C05454=1097.638,130.250,436.850,176.760,16.481,152.162
C05455=1097.644,130.499,436.829,176.762,16.481,152.162
C05456=1097.649,130.749,436.810,176.765,16.482,152.161
C05457=1097.656,130.998,436.790,176.768,16.482,152.161
C05458=1097.661,131.248,436.771,176.771,16.482,152.160
C05459=1097.667,131.496,436.751,176.774,16.482,152.159
C05460=1097.673,131.745,436.730,176.777,16.482,152.159
C05461=1097.678,131.995,436.711,176.780,16.482,152.158
C05462=1097.684,132.244,436.691,176.783,16.483,152.158
C05463=1097.690,132.493,436.671,176.785,16.483,152.157
C05464=1097.695,132.742,436.651,176.789,16.483,152.157
C05465=1097.701,132.991,436.631,176.792,16.484,152.156
C05466=1097.706,133.241,436.611,176.794,16.484,152.156
C05467=1097.712,133.490,436.591,176.798,16.484,152.155
C05468=1097.718,133.738,436.571,176.801,16.484,152.155
C05469=1097.724,133.988,436.551,176.803,16.485,152.154
C05470=1097.729,134.237,436.532,176.806,16.485,152.154
C05471=1097.734,134.486,436.511,176.810,16.485,152.153
C05472=1097.740,134.735,436.491,176.812,16.485,152.152
C05473=1097.746,134.984,436.472,176.815,16.485,152.152
C05474=1097.751,135.234,436.451,176.819,16.486,152.151
C05475=1097.757,135.482,436.431,176.821,16.486,152.151
C05476=1097.763,135.731,436.411,176.824,16.486,152.150
C05477=1097.768,135.981,436.392,176.828,16.486,152.150
C05478=1097.774,136.230,436.371,176.830,16.486,152.149
C05479=1097.780,136.479,436.351,176.833,16.487,152.149
C05480=1097.786,136.728,436.331,176.836,16.487,152.148
C05481=1097.791,136.977,436.311,176.839,16.487,152.147
C05482=1097.797,137.226,436.291,176.842,16.488,152.147
C05483=1097.802,137.475,436.271,176.845,16.488,152.146
C05484=1097.808,137.724,436.251,176.848,16.488,152.146
C05485=1097.814,137.974,436.230,176.851,16.488,152.145
C05486=1097.820,138.223,436.210,176.854,16.489,152.145
C05487=1097.825,138.472,436.189,176.857,16.488,152.144
C05488=1097.831,138.721,436.169,176.860,16.489,152.143
C05489=1097.836,138.970,436.150,176.863,16.489,152.143
C05490=1097.842,139.219,436.130,176.866,16.489,152.142
C05491=1097.847,139.468,436.109,176.869,16.489,152.142
C05492=1097.853,139.717,436.089,176.872,16.490,152.141
C05493=1097.858,139.966,436.069,176.875,16.489,152.141
C05494=1097.864,140.216,436.048,176.878,16.490,152.140
C05495=1097.870,140.465,436.028,176.881,16.490,152.139
C05496=1097.875,140.714,436.007,176.884,16.490,152.139
C05497=1097.881,140.963,435.987,176.887,16.490,152.138
C05498=1097.887,141.212,435.967,176.890,16.490,152.138
C05499=1097.892,141.461,435.946,176.893,16.490,152.137
C05500=1097.898,141.710,435.926,176.896,16.491,152.137
C05501=1097.903,141.959,435.906,176.899,16.491,152.136
C05502=1097.909,142.209,435.885,176.902,16.491,152.135
C05503=1097.915,142.458,435.865,176.905,16.491,152.135
C05504=1097.920,142.707,435.844,176.908,16.492,152.134
C05505=1097.926,142.956,435.824,176.912,16.492,152.134
C05506=1097.932,143.205,435.804,176.914,16.492,152.133
C05507=1097.937,143.454,435.783,176.917,16.492,152.133
C05508=1097.944,143.729,435.760,176.921,16.492,152.132
C05509=1097.950,144.003,435.738,176.924,16.492,152.131
C05510=1097.956,144.278,435.714,176.928,16.492,152.130
C05511=1097.962,144.552,435.692,176.931,16.493,152.130
C05512=1097.967,144.801,435.671,176.934,16.493,152.129
C05513=1097.973,145.050,435.652,176.937,16.493,152.129
C05514=1097.979,145.300,435.631,176.940,16.493,152.128
C05515=1097.985,145.549,435.610,176.943,16.493,152.128
C05516=1097.990,145.798,435.590,176.946,16.493,152.127
C05517=1097.996,146.046,435.569,176.949,16.493,152.126
C05518=1098.001,146.295,435.548,176.953,16.494,152.126
C05519=1098.007,146.545,435.527,176.955,16.493,152.125
C05520=1098.013,146.794,435.507,176.959,16.494,152.125
C05521=1098.019,147.043,435.487,176.962,16.494,152.124
C05522=1098.024,147.291,435.466,176.964,16.494,152.123
C05523=1098.030,147.541,435.445,176.968,16.494,152.123
C05524=1098.035,147.790,435.424,176.971,16.494,152.122
C05525=1098.041,148.039,435.404,176.974,16.494,152.122
C05526=1098.047,148.288,435.383,176.977,16.494,152.121
C05527=1098.053,148.537,435.362,176.980,16.494,152.120
C05528=1098.058,148.787,435.341,176.984,16.495,152.120
C05529=1098.063,149.035,435.320,176.986,16.494,152.119
C05530=1098.069,149.285,435.299,176.989,16.495,152.119
C05531=1098.075,149.534,435.279,176.993,16.495,152.118
C05532=1098.081,149.782,435.258,176.995,16.495,152.117
C05533=1098.086,150.031,435.237,176.999,16.495,152.117
C05534=1098.092,150.281,435.217,177.002,16.495,152.116
C05535=1098.097,150.530,435.195,177.005,16.495,152.115
C05536=1098.103,150.779,435.175,177.008,16.495,152.115
C05537=1098.108,151.028,435.154,177.012,16.495,152.114
C05538=1098.114,151.277,435.132,177.015,16.496,152.114
C05539=1098.119,151.526,435.112,177.017,16.495,152.113
C05540=1098.125,151.775,435.091,177.021,16.496,152.112
C05541=1098.131,152.025,435.070,177.024,16.496,152.112
C05542=1098.137,152.273,435.049,177.027,16.495,152.111
C05543=1098.142,152.522,435.029,177.030,16.495,152.110
C05544=1098.148,152.772,435.008,177.033,16.496,152.110
C05545=1098.154,153.020,434.986,177.037,16.496,152.109
C05546=1098.159,153.269,434.966,177.039,16.496,152.109
C05547=1098.165,153.519,434.944,177.043,16.496,152.108
C05548=1098.170,153.768,434.924,177.046,16.496,152.107
C05549=1098.176,154.016,434.902,177.049,16.496,152.107
C05550=1098.182,154.266,434.881,177.052,16.496,152.106
C05551=1098.187,154.515,434.860,177.055,16.496,152.105
C05552=1098.193,154.763,434.839,177.059,16.496,152.105
C05553=1098.199,155.013,434.818,177.061,16.496,152.104
C05554=1098.204,155.261,434.797,177.065,16.496,152.104
C05555=1098.210,155.511,434.776,177.068,16.497,152.103
C05556=1098.216,155.760,434.754,177.071,16.496,152.102
C05557=1098.221,156.009,434.734,177.074,16.496,152.102
C05558=1098.227,156.258,434.712,177.078,16.496,152.101
C05559=1098.232,156.507,434.690,177.081,16.497,152.100
C05560=1098.238,156.757,434.670,177.084,16.496,152.100
C05561=1098.244,157.005,434.648,177.087,16.497,152.099
C05562=1098.249,157.254,434.627,177.090,16.496,152.098
C05563=1098.255,157.504,434.606,177.094,16.497,152.098
C05564=1098.261,157.752,434.585,177.096,16.496,152.097
C05565=1098.267,158.001,434.563,177.100,16.497,152.097
C05566=1098.272,158.250,434.543,177.103,16.497,152.096
C05567=1098.277,158.499,434.521,177.106,16.496,152.095
C05568=1098.283,158.748,434.499,177.109,16.496,152.095
C05569=1098.288,158.997,434.479,177.112,16.497,152.094
C05570=1098.294,159.247,434.457,177.116,16.497,152.093
C05571=1098.300,159.495,434.436,177.118,16.497,152.093
C05572=1098.306,159.770,434.412,177.122,16.497,152.092
C05573=1098.312,160.044,434.389,177.126,16.496,152.091
C05574=1098.319,160.318,434.365,177.129,16.496,152.091
C05575=1098.325,160.592,434.341,177.133,16.496,152.090
C05576=1098.331,160.842,434.320,177.136,16.496,152.089
C05577=1098.335,161.090,434.299,177.139,16.497,152.089
C05578=1098.342,161.340,434.277,177.143,16.497,152.088
C05579=1098.347,161.588,434.256,177.146,16.497,152.087
C05580=1098.353,161.837,434.234,177.149,16.496,152.087
C05581=1098.358,162.086,434.212,177.152,16.497,152.086
C05582=1098.364,162.336,434.191,177.156,16.497,152.085
C05583=1098.370,162.585,434.170,177.158,16.497,152.085
C05584=1098.374,162.833,434.148,177.162,16.497,152.084
C05585=1098.381,163.083,434.126,177.165,16.497,152.083
C05586=1098.385,163.331,434.105,177.169,16.497,152.083
C05587=1098.392,163.581,434.083,177.171,16.496,152.082
C05588=1098.396,163.829,434.061,177.175,16.497,152.081
C05589=1098.403,164.079,434.039,177.178,16.497,152.081
C05590=1098.408,164.327,434.018,177.181,16.497,152.080
C05591=1098.413,164.577,433.996,177.184,16.497,152.079
C05592=1098.419,164.825,433.975,177.188,16.497,152.079
C05593=1098.424,165.074,433.953,177.191,16.497,152.078
C05594=1098.430,165.323,433.931,177.195,16.497,152.077
C05595=1098.435,165.572,433.909,177.198,16.497,152.077
C05596=1098.441,165.821,433.888,177.201,16.497,152.076
C05597=1098.446,166.070,433.866,177.204,16.497,152.075
C05598=1098.452,166.319,433.844,177.207,16.497,152.075
C05599=1098.457,166.568,433.822,177.211,16.497,152.074
C05600=1098.463,166.817,433.801,177.214,16.496,152.073
C05601=1098.469,167.066,433.779,177.217,16.497,152.073
C05602=1098.474,167.315,433.757,177.221,16.497,152.072
C05603=1098.480,167.564,433.736,177.224,16.497,152.071
C05604=1098.485,167.813,433.714,177.227,16.497,152.071
C05605=1098.491,168.062,433.692,177.230,16.497,152.070
C05606=1098.496,168.311,433.670,177.234,16.497,152.069
C05607=1098.502,168.560,433.649,177.237,16.497,152.069
C05608=1098.507,168.809,433.626,177.240,16.496,152.068
C05609=1098.513,169.058,433.604,177.243,16.496,152.067
C05610=1098.519,169.307,433.582,177.247,16.496,152.067
C05611=1098.524,169.556,433.560,177.250,16.497,152.066
C05612=1098.530,169.805,433.539,177.254,16.497,152.065
C05613=1098.535,170.054,433.517,177.256,16.496,152.065
C05614=1098.541,170.303,433.494,177.260,16.496,152.064
C05615=1098.546,170.552,433.473,177.263,16.496,152.063
C05616=1098.552,170.801,433.451,177.267,16.496,152.063
C05617=1098.558,171.050,433.429,177.269,16.496,152.062
C05618=1098.563,171.298,433.407,177.273,16.496,152.061
C05619=1098.569,171.548,433.384,177.276,16.496,152.061
C05620=1098.574,171.797,433.362,177.280,16.496,152.060
C05621=1098.580,172.046,433.341,177.283,16.496,152.059
C05622=1098.586,172.295,433.318,177.286,16.495,152.059
C05623=1098.592,172.544,433.296,177.290,16.495,152.058
C05624=1098.597,172.793,433.274,177.293,16.495,152.057
C05625=1098.602,173.042,433.252,177.297,16.495,152.056
C05626=1098.608,173.291,433.230,177.299,16.495,152.056
C05627=1098.613,173.540,433.208,177.303,16.495,152.055
C05628=1098.620,173.788,433.186,177.306,16.495,152.054
C05629=1098.625,174.038,433.163,177.310,16.495,152.054
C05630=1098.630,174.287,433.142,177.313,16.495,152.053
C05631=1098.636,174.535,433.119,177.316,16.495,152.052
C05632=1098.642,174.785,433.097,177.320,16.495,152.052
C05633=1098.647,175.033,433.074,177.323,16.494,152.051
C05634=1098.653,175.282,433.053,177.327,16.494,152.050
C05635=1098.659,175.532,433.031,177.329,16.494,152.049
C05636=1098.665,175.805,433.006,177.334,16.494,152.049
C05637=1098.671,176.079,432.981,177.338,16.494,152.048
C05638=1098.678,176.353,432.957,177.341,16.494,152.047
C05639=1098.683,176.626,432.932,177.345,16.493,152.046
C05640=1098.689,176.876,432.911,177.349,16.493,152.045
C05641=1098.695,177.124,432.888,177.351,16.493,152.045
C05642=1098.700,177.374,432.865,177.355,16.493,152.044
C05643=1098.707,177.623,432.843,177.358,16.493,152.043
C05644=1098.712,177.871,432.820,177.362,16.493,152.043
C05645=1098.718,178.120,432.798,177.365,16.492,152.042
C05646=1098.723,178.369,432.775,177.368,16.492,152.041
C05647=1098.729,178.618,432.754,177.372,16.492,152.040
C05648=1098.735,178.867,432.731,177.375,16.492,152.040
C05649=1098.740,179.116,432.709,177.379,16.492,152.039
C05650=1098.746,179.365,432.686,177.382,16.491,152.038
C05651=1098.752,179.614,432.664,177.385,16.491,152.038
C05652=1098.758,179.863,432.641,177.389,16.491,152.037
C05653=1098.763,180.112,432.618,177.392,16.491,152.036
C05654=1098.770,180.361,432.596,177.396,16.491,152.035
C05655=1098.775,180.609,432.574,177.399,16.490,152.035
C05656=1098.780,180.858,432.551,177.402,16.490,152.034
C05657=1098.786,181.107,432.528,177.406,16.490,152.033
C05658=1098.792,181.356,432.507,177.410,16.490,152.032
C05659=1098.798,181.605,432.484,177.413,16.490,152.032
C05660=1098.804,181.854,432.461,177.416,16.490,152.031
C05661=1098.809,182.103,432.438,177.420,16.489,152.030
C05662=1098.814,182.352,432.416,177.423,16.489,152.029
C05663=1098.821,182.600,432.394,177.427,16.489,152.029
C05664=1098.826,182.849,432.371,177.430,16.489,152.028
C05665=1098.832,183.098,432.348,177.433,16.489,152.027
C05666=1098.838,183.348,432.325,177.437,16.488,152.026
C05667=1098.843,183.597,432.302,177.440,16.488,152.026
C05668=1098.850,183.845,432.280,177.444,16.488,152.025
C05669=1098.856,184.094,432.257,177.448,16.488,152.024
C05670=1098.861,184.343,432.234,177.451,16.487,152.023
C05671=1098.867,184.592,432.211,177.454,16.487,152.023
C05672=1098.872,184.841,432.189,177.458,16.487,152.022
C05673=1098.878,185.090,432.166,177.461,16.487,152.021
C05674=1098.884,185.339,432.143,177.465,16.487,152.020
C05675=1098.889,185.587,432.121,177.469,16.487,152.020
C05676=1098.895,185.836,432.098,177.471,16.486,152.019
C05677=1098.900,186.085,432.075,177.475,16.486,152.018
C05678=1098.906,186.334,432.052,177.478,16.486,152.017
C05679=1098.912,186.583,432.029,177.482,16.486,152.017
C05680=1098.918,186.832,432.006,177.486,16.486,152.016
C05681=1098.923,187.081,431.983,177.489,16.486,152.015
C05682=1098.927,187.330,431.960,177.492,16.485,152.015
C05683=1098.933,187.579,431.938,177.496,16.485,152.014
C05684=1098.939,187.828,431.915,177.499,16.485,152.013
C05685=1098.945,188.077,431.892,177.503,16.485,152.012
C05686=1098.950,188.326,431.869,177.506,16.485,152.012
C05687=1098.956,188.574,431.846,177.510,16.485,152.011
C05688=1098.961,188.824,431.822,177.513,16.484,152.010
C05689=1098.967,189.073,431.799,177.516,16.484,152.009
C05690=1098.973,189.321,431.776,177.520,16.484,152.009
C05691=1098.979,189.570,431.753,177.523,16.484,152.008
C05692=1098.984,189.818,431.730,177.527,16.484,152.007
C05693=1098.989,190.067,431.707,177.531,16.483,152.006
C05694=1098.994,190.316,431.684,177.534,16.483,152.006
C05695=1099.000,190.565,431.661,177.537,16.483,152.005
C05696=1099.006,190.814,431.638,177.541,16.483,152.004
C05697=1099.012,191.063,431.615,177.545,16.482,152.003
C05698=1099.017,191.312,431.591,177.548,16.482,152.003
C05699=1099.022,191.561,431.568,177.552,16.482,152.002
C05700=1099.029,191.834,431.542,177.555,16.482,152.001
C05701=1099.035,192.108,431.517,177.559,16.482,152.000
C05702=1099.041,192.381,431.491,177.563,16.482,151.999
C05703=1099.047,192.654,431.465,177.567,16.481,151.998
C05704=1099.053,192.903,431.443,177.570,16.481,151.998
C05705=1099.059,193.152,431.420,177.574,16.481,151.997
C05706=1099.064,193.401,431.396,177.578,16.481,151.996
C05707=1099.070,193.650,431.373,177.581,16.481,151.995
C05708=1099.076,193.899,431.349,177.584,16.480,151.995
C05709=1099.081,194.147,431.326,177.588,16.480,151.994
C05710=1099.086,194.397,431.303,177.591,16.480,151.993
C05711=1099.092,194.645,431.279,177.595,16.479,151.992
C05712=1099.098,194.894,431.256,177.599,16.479,151.992
C05713=1099.103,195.143,431.233,177.602,16.479,151.991
C05714=1099.109,195.391,431.209,177.606,16.479,151.990
C05715=1099.115,195.641,431.186,177.609,16.478,151.989
C05716=1099.120,195.890,431.162,177.613,16.478,151.988
C05717=1099.126,196.138,431.139,177.616,16.478,151.988
C05718=1099.132,196.387,431.116,177.620,16.478,151.987
C05719=1099.137,196.637,431.092,177.623,16.477,151.986
C05720=1099.143,196.885,431.068,177.627,16.478,151.985
C05721=1099.149,197.134,431.046,177.631,16.477,151.984
C05722=1099.154,197.382,431.021,177.634,16.477,151.984
C05723=1099.160,197.631,430.998,177.637,16.476,151.983
C05724=1099.166,197.881,430.975,177.641,16.476,151.982
C05725=1099.172,198.129,430.951,177.645,16.476,151.981
C05726=1099.177,198.378,430.928,177.648,16.476,151.981
C05727=1099.183,198.627,430.904,177.652,16.475,151.980
C05728=1099.188,198.876,430.881,177.656,16.475,151.979
C05729=1099.194,199.124,430.857,177.660,16.475,151.978
C05730=1099.199,199.373,430.833,177.662,16.474,151.977
C05731=1099.206,199.622,430.809,177.666,16.474,151.977
C05732=1099.212,199.871,430.786,177.670,16.474,151.976
C05733=1099.217,200.120,430.762,177.674,16.473,151.975
C05734=1099.223,200.368,430.739,177.677,16.473,151.974
C05735=1099.228,200.617,430.715,177.681,16.473,151.973
C05736=1099.235,200.866,430.691,177.684,16.473,151.973
C05737=1099.240,201.115,430.668,177.688,16.473,151.972
C05738=1099.246,201.364,430.644,177.691,16.472,151.971
C05739=1099.252,201.612,430.620,177.695,16.472,151.970
C05740=1099.257,201.862,430.596,177.699,16.471,151.969
C05741=1099.263,202.110,430.573,177.702,16.471,151.969
C05742=1099.269,202.359,430.548,177.706,16.471,151.968
C05743=1099.274,202.608,430.525,177.710,16.470,151.967
C05744=1099.280,202.856,430.501,177.713,16.470,151.966
C05745=1099.286,203.105,430.477,177.717,16.470,151.965
C05746=1099.291,203.354,430.453,177.720,16.469,151.965
C05747=1099.297,203.603,430.430,177.724,16.469,151.964
C05748=1099.303,203.851,430.406,177.727,16.469,151.963
C05749=1099.308,204.100,430.382,177.731,16.469,151.962
C05750=1099.314,204.349,430.358,177.735,16.469,151.962
C05751=1099.320,204.598,430.334,177.739,16.468,151.961
C05752=1099.325,204.847,430.309,177.742,16.468,151.960
C05753=1099.331,205.095,430.287,177.746,16.468,151.959
C05754=1099.337,205.345,430.262,177.750,16.468,151.958
C05755=1099.342,205.593,430.238,177.753,16.467,151.957
C05756=1099.348,205.842,430.214,177.756,16.466,151.957
C05757=1099.353,206.090,430.190,177.760,16.466,151.956
C05758=1099.359,206.340,430.166,177.764,16.466,151.955
C05759=1099.365,206.588,430.142,177.767,16.466,151.954
C05760=1099.370,206.837,430.118,177.771,16.466,151.953
C05761=1099.375,207.086,430.094,177.775,16.465,151.953
C05762=1099.382,207.335,430.070,177.778,16.465,151.952
C05763=1099.387,207.583,430.045,177.782,16.465,151.951
C05764=1099.410,208.592,429.948,177.824,16.478,151.946
C05765=1099.419,208.961,429.911,177.829,16.479,151.945
C05766=1099.427,209.331,429.875,177.833,16.480,151.944
C05767=1099.436,209.701,429.839,177.839,16.480,151.943
C05768=1099.444,210.070,429.803,177.844,16.482,151.942
C05769=1099.450,210.320,429.778,177.847,16.482,151.941
C05770=1099.455,210.568,429.754,177.851,16.482,151.941
C05771=1099.461,210.818,429.729,177.855,16.483,151.940
C05772=1099.466,211.066,429.704,177.858,16.484,151.940
C05773=1099.472,211.314,429.680,177.861,16.484,151.939
C05774=1099.478,211.563,429.656,177.864,16.485,151.939
C05775=1099.483,211.812,429.631,177.868,16.485,151.938
C05776=1099.489,212.061,429.607,177.872,16.486,151.938
C05777=1099.494,212.309,429.582,177.875,16.486,151.937
C05778=1099.500,212.558,429.557,177.878,16.487,151.936
C05779=1099.506,212.807,429.533,177.882,16.487,151.936
C05780=1099.511,213.056,429.509,177.885,16.488,151.935
C05781=1099.517,213.304,429.483,177.889,16.489,151.935
C05782=1099.522,213.553,429.459,177.892,16.489,151.934
C05783=1099.528,213.802,429.434,177.895,16.490,151.934
C05784=1099.534,214.051,429.410,177.899,16.490,151.933
C05785=1099.539,214.299,429.385,177.903,16.492,151.932
C05786=1099.545,214.548,429.361,177.906,16.492,151.932
C05787=1099.550,214.797,429.336,177.909,16.493,151.931
C05788=1099.557,215.045,429.311,177.912,16.493,151.931
C05789=1099.561,215.294,429.286,177.916,16.494,151.930
C05790=1099.567,215.543,429.261,177.920,16.494,151.930
C05791=1099.573,215.792,429.236,177.923,16.495,151.929
C05792=1099.579,216.041,429.212,177.926,16.495,151.928
C05793=1099.584,216.289,429.187,177.930,16.496,151.928
C05794=1099.590,216.538,429.162,177.934,16.497,151.927
C05795=1099.596,216.786,429.137,177.937,16.497,151.927
C05796=1099.601,217.036,429.112,177.940,16.498,151.926
C05797=1099.606,217.284,429.087,177.943,16.498,151.926
C05798=1099.612,217.533,429.062,177.947,16.499,151.925
C05799=1099.618,217.782,429.038,177.951,16.500,151.925
C05800=1099.624,218.030,429.013,177.954,16.500,151.924
C05801=1099.628,218.279,428.988,177.957,16.501,151.923
C05802=1099.635,218.528,428.963,177.961,16.502,151.923
C05803=1099.640,218.776,428.938,177.965,16.502,151.922
C05804=1099.646,219.025,428.913,177.968,16.503,151.922
C05805=1099.652,219.273,428.888,177.971,16.503,151.921
C05806=1099.657,219.523,428.863,177.975,16.504,151.921
C05807=1099.663,219.771,428.838,177.978,16.505,151.920
C05808=1099.668,220.020,428.813,177.982,16.505,151.919
C05809=1099.675,220.269,428.788,177.985,16.506,151.919
C05810=1099.679,220.517,428.762,177.989,16.507,151.918
C05811=1099.685,220.766,428.738,177.992,16.507,151.918
C05812=1099.692,221.015,428.712,177.995,16.508,151.917
C05813=1099.697,221.263,428.687,177.999,16.508,151.917
C05814=1099.702,221.512,428.662,178.003,16.509,151.916
C05815=1099.708,221.760,428.637,178.006,16.510,151.915
C05816=1099.714,222.009,428.612,178.009,16.510,151.915
C05817=1099.723,222.383,428.574,178.014,16.511,151.914
C05818=1099.731,222.757,428.536,178.020,16.512,151.913
C05819=1099.739,223.131,428.499,178.025,16.514,151.913
C05820=1099.748,223.504,428.460,178.030,16.514,151.912
C05821=1099.753,223.753,428.435,178.033,16.515,151.911
C05822=1099.759,224.001,428.410,178.037,16.516,151.910
C05823=1099.764,224.250,428.385,178.041,16.517,151.910
C05824=1099.770,224.498,428.359,178.044,16.517,151.909
C05825=1099.775,224.747,428.333,178.047,16.518,151.909
C05826=1099.781,224.995,428.308,178.051,16.519,151.908
C05827=1099.786,225.245,428.283,178.054,16.519,151.908
C05828=1099.792,225.494,428.258,178.058,16.520,151.907
C05829=1099.797,225.742,428.232,178.062,16.521,151.907
C05830=1099.804,225.991,428.207,178.065,16.521,151.906
C05831=1099.810,226.239,428.181,178.068,16.522,151.906
C05832=1099.815,226.487,428.156,178.071,16.522,151.905
C05833=1099.821,226.736,428.131,178.075,16.524,151.904
C05834=1099.826,226.985,428.105,178.079,16.524,151.904
C05835=1099.832,227.234,428.079,178.082,16.525,151.903
C05836=1099.837,227.482,428.054,178.086,16.526,151.903
C05837=1099.843,227.731,428.028,178.089,16.526,151.902
C05838=1099.849,227.980,428.002,178.093,16.526,151.902
C05839=1099.854,228.228,427.977,178.097,16.527,151.901
C05840=1099.860,228.477,427.952,178.100,16.528,151.900
C05841=1099.866,228.726,427.926,178.103,16.528,151.900
C05842=1099.872,228.974,427.900,178.107,16.530,151.899
C05843=1099.877,229.223,427.875,178.110,16.530,151.899
C05844=1099.883,229.471,427.849,178.114,16.531,151.898
C05845=1099.888,229.720,427.823,178.117,16.531,151.898
C05846=1099.895,229.969,427.798,178.121,16.532,151.897
C05847=1099.900,230.218,427.772,178.124,16.533,151.897
C05848=1099.905,230.466,427.747,178.127,16.533,151.896
C05849=1099.911,230.715,427.721,178.131,16.534,151.896
C05850=1099.917,230.963,427.695,178.135,16.535,151.895
C05851=1099.922,231.212,427.669,178.138,16.536,151.894
C05852=1099.928,231.460,427.644,178.142,16.537,151.894
C05853=1099.933,231.709,427.618,178.145,16.537,151.893
C05854=1099.939,231.958,427.592,178.148,16.538,151.893
C05855=1099.944,232.207,427.566,178.152,16.539,151.892
C05856=1099.951,232.455,427.540,178.156,16.539,151.892
C05857=1099.956,232.703,427.514,178.159,16.540,151.891
C05858=1099.961,232.952,427.488,178.163,16.541,151.891
C05859=1099.967,233.201,427.463,178.166,16.542,151.890
C05860=1099.973,233.449,427.436,178.169,16.542,151.890
C05861=1099.979,233.698,427.410,178.173,16.543,151.889
C05862=1099.984,233.947,427.385,178.176,16.544,151.888
C05863=1099.990,234.195,427.359,178.180,16.544,151.888
C05864=1099.995,234.444,427.333,178.184,16.545,151.887
C05865=1100.001,234.693,427.307,178.187,16.546,151.887
C05866=1100.007,234.941,427.280,178.191,16.547,151.886
C05867=1100.012,235.190,427.254,178.194,16.548,151.886
C05868=1100.018,235.439,427.228,178.197,16.549,151.885
C05869=1100.025,235.803,427.190,178.203,16.549,151.884
C05870=1100.034,236.169,427.152,178.208,16.551,151.884
C05871=1100.042,236.534,427.113,178.213,16.552,151.883
C05872=1100.050,236.899,427.075,178.218,16.553,151.882
C05873=1100.056,237.148,427.049,178.221,16.554,151.882
C05874=1100.062,237.396,427.023,178.225,16.555,151.881
C05875=1100.068,237.645,426.997,178.228,16.556,151.881
C05876=1100.074,237.893,426.970,178.232,16.557,151.880
C05877=1100.079,238.142,426.944,178.236,16.557,151.880
C05878=1100.084,238.390,426.918,178.239,16.558,151.879
C05879=1100.090,238.639,426.892,178.243,16.559,151.878
C05880=1100.096,238.887,426.866,178.246,16.559,151.878
C05881=1100.101,239.136,426.840,178.249,16.560,151.877
C05882=1100.107,239.384,426.813,178.253,16.561,151.877
C05883=1100.112,239.633,426.787,178.256,16.562,151.876
C05884=1100.118,239.882,426.760,178.260,16.563,151.876
C05885=1100.124,240.130,426.734,178.264,16.563,151.875
C05886=1100.129,240.379,426.708,178.267,16.564,151.875
C05887=1100.135,240.628,426.681,178.271,16.565,151.874
C05888=1100.141,240.877,426.655,178.274,16.566,151.874
C05889=1100.146,241.125,426.629,178.277,16.567,151.873
C05890=1100.152,241.373,426.602,178.281,16.568,151.873
C05891=1100.158,241.622,426.575,178.284,16.568,151.872
C05892=1100.163,241.871,426.549,178.288,16.569,151.872
C05893=1100.169,242.119,426.523,178.292,16.570,151.871
C05894=1100.175,242.367,426.496,178.295,16.570,151.870
C05895=1100.180,242.616,426.470,178.299,16.572,151.870
C05896=1100.186,242.865,426.443,178.302,16.572,151.869
C05897=1100.192,243.113,426.417,178.306,16.573,151.869
C05898=1100.198,243.361,426.390,178.309,16.574,151.868
C05899=1100.203,243.610,426.364,178.312,16.575,151.868
C05900=1100.209,243.859,426.338,178.316,16.576,151.867
C05901=1100.214,244.107,426.310,178.319,16.576,151.867
C05902=1100.220,244.356,426.284,178.323,16.578,151.866
C05903=1100.225,244.604,426.257,178.327,16.578,151.866
C05904=1100.231,244.852,426.230,178.331,16.579,151.865
C05905=1100.237,245.101,426.204,178.334,16.580,151.865
C05906=1100.242,245.350,426.177,178.337,16.581,151.864
C05907=1100.248,245.598,426.151,178.341,16.582,151.864
C05908=1100.253,245.847,426.124,178.344,16.583,151.863
C05909=1100.259,246.095,426.097,178.348,16.584,151.863
C05910=1100.265,246.344,426.070,178.351,16.585,151.862
C05911=1100.271,246.593,426.043,178.355,16.586,151.862
C05912=1100.276,246.841,426.016,178.358,16.586,151.861
C05913=1100.282,247.090,425.990,178.361,16.587,151.861
C05914=1100.288,247.338,425.963,178.365,16.588,151.860
C05915=1100.293,247.587,425.936,178.369,16.589,151.860
C05916=1100.299,247.835,425.909,178.372,16.590,151.859
C05917=1100.304,248.083,425.883,178.376,16.591,151.859
C05918=1100.309,248.332,425.855,178.380,16.592,151.858
C05919=1100.315,248.580,425.829,178.383,16.593,151.858
C05920=1100.320,248.829,425.801,178.387,16.594,151.857
C05921=1100.328,249.187,425.763,178.391,16.595,151.857
C05922=1100.337,249.545,425.724,178.396,16.596,151.856
C05923=1100.344,249.904,425.685,178.401,16.597,151.855
C05924=1100.353,250.263,425.646,178.406,16.599,151.854
C05925=1100.358,250.511,425.618,178.410,16.600,151.854
C05926=1100.364,250.760,425.592,178.413,16.601,151.853
C05927=1100.370,251.008,425.565,178.417,16.602,151.853
C05928=1100.375,251.256,425.537,178.420,16.603,151.852
C05929=1100.381,251.504,425.511,178.424,16.604,151.852
C05930=1100.386,251.753,425.483,178.427,16.605,151.851
C05931=1100.392,252.001,425.457,178.431,16.606,151.851
C05932=1100.397,252.251,425.429,178.434,16.607,151.850
C05933=1100.403,252.498,425.402,178.438,16.608,151.850
C05934=1100.408,252.747,425.374,178.441,16.609,151.849
C05935=1100.414,252.996,425.348,178.445,16.610,151.849
C05936=1100.419,253.244,425.321,178.449,16.610,151.848
C05937=1100.426,253.493,425.293,178.452,16.612,151.848
C05938=1100.431,253.741,425.266,178.456,16.613,151.847
C05939=1100.437,253.990,425.239,178.459,16.613,151.847
C05940=1100.442,254.238,425.211,178.462,16.615,151.847
C05941=1100.448,254.486,425.184,178.466,16.615,151.846
C05942=1100.454,254.735,425.156,178.470,16.616,151.845
C05943=1100.459,254.983,425.129,178.473,16.617,151.845
C05944=1100.464,255.232,425.102,178.477,16.619,151.845
C05945=1100.471,255.480,425.075,178.480,16.619,151.844
C05946=1100.476,255.729,425.047,178.484,16.620,151.843
C05947=1100.482,255.977,425.019,178.487,16.621,151.843
C05948=1100.487,256.225,424.992,178.491,16.622,151.843
C05949=1100.492,256.474,424.965,178.494,16.623,151.842
C05950=1100.499,256.722,424.938,178.498,16.624,151.841
C05951=1100.504,256.971,424.910,178.501,16.625,151.841
C05952=1100.510,257.219,424.883,178.505,16.626,151.841
C05953=1100.516,257.468,424.855,178.508,16.627,151.840
C05954=1100.521,257.716,424.827,178.512,16.629,151.840
C05955=1100.527,257.964,424.800,178.515,16.629,151.839
C05956=1100.532,258.213,424.773,178.519,16.630,151.839
C05957=1100.538,258.461,424.744,178.522,16.631,151.838
C05958=1100.544,258.710,424.718,178.526,16.632,151.838
C05959=1100.549,258.958,424.690,178.529,16.633,151.837
C05960=1100.556,259.206,424.662,178.533,16.634,151.837
C05961=1100.561,259.455,424.635,178.536,16.635,151.836
C05962=1100.566,259.703,424.607,178.540,16.636,151.836
C05963=1100.573,259.952,424.580,178.543,16.637,151.835
C05964=1100.578,260.200,424.552,178.547,16.638,151.835
C05965=1100.584,260.449,424.524,178.550,16.639,151.834
C05966=1100.590,260.697,424.496,178.554,16.640,151.834
C05967=1100.595,260.945,424.469,178.558,16.641,151.833
C05968=1100.601,261.194,424.441,178.561,16.642,151.833
C05969=1100.607,261.442,424.413,178.565,16.643,151.832
C05970=1100.613,261.691,424.386,178.569,16.644,151.832
C05971=1100.618,261.939,424.358,178.571,16.645,151.831
C05972=1100.623,262.187,424.330,178.575,16.646,151.831
C05973=1100.633,262.543,424.290,178.581,16.648,151.830
C05974=1100.640,262.898,424.251,178.586,16.649,151.829
C05975=1100.649,263.254,424.210,178.591,16.650,151.829
C05976=1100.657,263.609,424.171,178.596,16.652,151.828
C05977=1100.663,263.858,424.142,178.599,16.653,151.828
C05978=1100.669,264.105,424.115,178.603,16.654,151.827
C05979=1100.675,264.354,424.087,178.607,16.655,151.827
C05980=1100.680,264.602,424.059,178.610,16.656,151.826
C05981=1100.686,264.852,424.031,178.614,16.657,151.826
C05982=1100.691,265.100,424.003,178.617,16.658,151.825
C05983=1100.697,265.348,423.975,178.621,16.659,151.825
C05984=1100.702,265.596,423.947,178.623,16.660,151.824
C05985=1100.708,265.844,423.919,178.627,16.662,151.824
C05986=1100.713,266.093,423.891,178.631,16.663,151.823
C05987=1100.719,266.341,423.863,178.634,16.664,151.823
C05988=1100.725,266.590,423.834,178.638,16.665,151.823
C05989=1100.730,266.838,423.806,178.641,16.666,151.822
C05990=1100.736,267.087,423.778,178.645,16.668,151.822
C05991=1100.741,267.335,423.750,178.648,16.668,151.821
C05992=1100.747,267.584,423.722,178.652,16.670,151.821
C05993=1100.753,267.832,423.694,178.656,16.671,151.820
C05994=1100.759,268.080,423.665,178.659,16.672,151.820
C05995=1100.764,268.328,423.637,178.663,16.673,151.819
C05996=1100.770,268.577,423.608,178.666,16.674,151.819
C05997=1100.776,268.825,423.580,178.670,16.675,151.818
C05998=1100.781,269.073,423.552,178.673,16.676,151.818
C05999=1100.787,269.321,423.524,178.677,16.678,151.818
C06000=1100.793,269.570,423.496,178.680,16.679,151.817
C06001=1100.798,269.818,423.467,178.684,16.680,151.817
C06002=1100.804,270.066,423.439,178.687,16.681,151.816
C06003=1100.810,270.314,423.411,178.691,16.682,151.816
C06004=1100.816,270.563,423.383,178.694,16.684,151.815
C06005=1100.821,270.811,423.355,178.697,16.684,151.815
C06006=1100.827,271.059,423.326,178.701,16.686,151.814
C06007=1100.833,271.307,423.298,178.705,16.687,151.814
C06008=1100.838,271.556,423.269,178.708,16.688,151.814
C06009=1100.843,271.804,423.240,178.712,16.690,151.813
C06010=1100.849,272.053,423.212,178.715,16.690,151.813
C06011=1100.855,272.301,423.183,178.719,16.692,151.812
C06012=1100.861,272.549,423.155,178.723,16.693,151.812
C06013=1100.867,272.798,423.126,178.726,16.694,151.811
C06014=1100.872,273.046,423.098,178.729,16.696,151.811
C06015=1100.878,273.294,423.069,178.733,16.696,151.811
C06016=1100.884,273.543,423.040,178.736,16.698,151.810
C06017=1100.889,273.791,423.012,178.740,16.699,151.810
C06018=1100.895,274.039,422.983,178.743,16.700,151.809
C06019=1100.900,274.287,422.955,178.747,16.702,151.809
C06020=1100.906,274.535,422.926,178.750,16.702,151.808
C06021=1100.912,274.784,422.898,178.754,16.704,151.808
C06022=1100.917,275.032,422.868,178.757,16.705,151.808
C06023=1100.923,275.281,422.840,178.761,16.706,151.807
C06024=1100.929,275.528,422.811,178.764,16.708,151.807
C06025=1100.936,275.887,422.770,178.769,16.710,151.806
C06026=1100.944,276.245,422.729,178.774,16.711,151.806
C06027=1100.953,276.603,422.687,178.780,16.713,151.805
C06028=1100.961,276.962,422.646,178.785,16.715,151.804
C06029=1100.966,277.210,422.616,178.788,16.716,151.804
C06030=1100.972,277.458,422.588,178.791,16.717,151.804
C06031=1100.979,277.707,422.559,178.795,16.719,151.803
C06032=1100.983,277.954,422.530,178.798,16.720,151.803
C06033=1100.989,278.203,422.501,178.802,16.721,151.802
C06034=1100.995,278.452,422.472,178.806,16.723,151.802
C06035=1101.001,278.699,422.443,178.809,16.724,151.802
C06036=1101.007,278.948,422.415,178.812,16.725,151.801
C06037=1101.012,279.196,422.385,178.816,16.727,151.801
C06038=1101.018,279.444,422.356,178.819,16.728,151.800
C06039=1101.023,279.692,422.327,178.823,16.729,151.800
C06040=1101.029,279.941,422.298,178.826,16.730,151.800
C06041=1101.034,280.188,422.269,178.830,16.732,151.799
C06042=1101.040,280.437,422.240,178.834,16.733,151.799
C06043=1101.047,280.685,422.211,178.837,16.734,151.798
C06044=1101.052,280.934,422.182,178.840,16.736,151.798
C06045=1101.057,281.181,422.153,178.844,16.737,151.797
C06046=1101.063,281.430,422.124,178.847,16.738,151.797
C06047=1101.068,281.678,422.094,178.851,16.740,151.797
C06048=1101.075,281.926,422.065,178.855,16.741,151.796
C06049=1101.079,282.175,422.037,178.858,16.742,151.796
C06050=1101.086,282.423,422.008,178.861,16.744,151.796
C06051=1101.091,282.671,421.978,178.865,16.745,151.795
C06052=1101.097,282.920,421.948,178.868,16.746,151.795
C06053=1101.102,283.167,421.920,178.872,16.748,151.794
C06054=1101.108,283.416,421.890,178.876,16.749,151.794
C06055=1101.114,283.664,421.861,178.878,16.750,151.794
C06056=1101.119,283.912,421.831,178.882,16.752,151.793
C06057=1101.124,284.160,421.802,178.886,16.754,151.793
C06058=1101.131,284.408,421.773,178.890,16.755,151.793
C06059=1101.136,284.656,421.743,178.892,16.756,151.792
C06060=1101.142,284.905,421.714,178.896,16.758,151.792
C06061=1101.147,285.152,421.685,178.900,16.760,151.791
C06062=1101.153,285.401,421.655,178.903,16.760,151.791
C06063=1101.158,285.649,421.626,178.907,16.762,151.791
C06064=1101.165,285.897,421.597,178.910,16.764,151.790
C06065=1101.170,286.146,421.567,178.913,16.765,151.790
C06066=1101.176,286.394,421.537,178.917,16.766,151.789
C06067=1101.181,286.642,421.509,178.921,16.768,151.789
C06068=1101.187,286.890,421.479,178.924,16.769,151.789
C06069=1101.193,287.138,421.449,178.927,16.770,151.788
C06070=1101.198,287.386,421.419,178.931,16.772,151.788
C06071=1101.204,287.634,421.390,178.935,16.774,151.788
C06072=1101.210,287.883,421.360,178.938,16.775,151.787
C06073=1101.215,288.131,421.331,178.941,16.776,151.787
C06074=1101.221,288.379,421.302,178.945,16.778,151.787
C06075=1101.227,288.627,421.272,178.948,16.779,151.786
C06076=1101.232,288.875,421.242,178.952,16.781,151.786
C06077=1101.241,289.243,421.198,178.957,16.783,151.785
C06078=1101.249,289.610,421.154,178.962,16.785,151.785
C06079=1101.258,289.978,421.110,178.968,16.787,151.784
C06080=1101.266,290.345,421.066,178.972,16.789,151.784
C06081=1101.272,290.593,421.036,178.976,16.791,151.783
C06082=1101.277,290.842,421.007,178.980,16.793,151.783
C06083=1101.283,291.090,420.976,178.983,16.794,151.783
C06084=1101.289,291.338,420.947,178.986,16.795,151.782
C06085=1101.295,291.586,420.918,178.990,16.797,151.782
C06086=1101.300,291.834,420.887,178.994,16.799,151.782
C06087=1101.306,292.083,420.858,178.996,16.800,151.781
C06088=1101.312,292.330,420.827,179.000,16.802,151.781
C06089=1101.317,292.579,420.798,179.004,16.803,151.781
C06090=1101.323,292.827,420.768,179.007,16.805,151.780
C06091=1101.329,293.075,420.738,179.010,16.806,151.780
C06092=1101.334,293.323,420.708,179.014,16.808,151.780
C06093=1101.340,293.571,420.678,179.018,16.809,151.779
C06094=1101.345,293.819,420.649,179.021,16.811,151.779
C06095=1101.351,294.067,420.618,179.024,16.812,151.779
C06096=1101.356,294.315,420.589,179.028,16.814,151.778
C06097=1101.362,294.563,420.558,179.031,16.816,151.778
C06098=1101.368,294.811,420.528,179.035,16.817,151.778
C06099=1101.373,295.059,420.498,179.038,16.818,151.777
C06100=1101.379,295.307,420.468,179.042,16.820,151.777
C06101=1101.385,295.556,420.438,179.045,16.822,151.777
C06102=1101.390,295.803,420.408,179.049,16.824,151.776
C06103=1101.396,296.051,420.378,179.053,16.825,151.776
C06104=1101.402,296.300,420.348,179.056,16.826,151.776
C06105=1101.408,296.548,420.317,179.059,16.828,151.775
C06106=1101.414,296.796,420.287,179.063,16.830,151.775
C06107=1101.420,297.045,420.257,179.066,16.832,151.775
C06108=1101.425,297.293,420.226,179.069,16.833,151.774
C06109=1101.430,297.540,420.196,179.073,16.835,151.774
C06110=1101.436,297.788,420.166,179.076,16.836,151.774
C06111=1101.442,298.037,420.136,179.080,16.838,151.773
C06112=1101.448,298.285,420.106,179.083,16.840,151.773
C06113=1101.453,298.532,420.075,179.086,16.841,151.773
C06114=1101.458,298.781,420.044,179.090,16.843,151.773
C06115=1101.464,299.029,420.015,179.093,16.845,151.772
C06116=1101.470,299.277,419.984,179.097,16.847,151.772
C06117=1101.475,299.525,419.953,179.101,16.849,151.772
C06118=1101.481,299.773,419.923,179.104,16.850,151.771
C06119=1101.487,300.021,419.893,179.107,16.852,151.771
C06120=1101.492,300.268,419.862,179.111,16.853,151.771
C06121=1101.497,300.517,419.832,179.114,16.855,151.771
C06122=1101.503,300.765,419.802,179.118,16.857,151.770
C06123=1101.509,301.013,419.771,179.121,16.859,151.770
C06124=1101.514,301.261,419.740,179.125,16.861,151.770
C06125=1101.520,301.509,419.710,179.127,16.862,151.770
C06126=1101.525,301.757,419.679,179.131,16.864,151.769
C06127=1101.531,302.005,419.649,179.134,16.866,151.769
C06128=1101.537,302.253,419.618,179.138,16.868,151.769
C06129=1101.545,302.634,419.571,179.143,16.871,151.768
C06130=1101.554,303.015,419.524,179.149,16.873,151.768
C06131=1101.562,303.397,419.477,179.154,16.876,151.767
C06132=1101.571,303.779,419.429,179.159,16.879,151.767
C06133=1101.576,304.026,419.399,179.163,16.881,151.767
C06134=1101.582,304.275,419.368,179.166,16.882,151.766
C06135=1101.588,304.523,419.337,179.169,16.884,151.766
C06136=1101.594,304.770,419.306,179.173,16.886,151.766
C06137=1101.599,305.018,419.275,179.176,16.888,151.766
C06138=1101.605,305.266,419.245,179.180,16.890,151.766
C06139=1101.610,305.514,419.214,179.183,16.891,151.765
C06140=1101.616,305.763,419.183,179.187,16.894,151.765
C06141=1101.621,306.011,419.153,179.190,16.895,151.765
C06142=1101.628,306.258,419.121,179.193,16.897,151.764
C06143=1101.633,306.506,419.091,179.196,16.899,151.764
C06144=1101.638,306.754,419.060,179.200,16.900,151.764
C06145=1101.644,307.003,419.029,179.204,16.902,151.764
C06146=1101.650,307.250,418.998,179.207,16.904,151.763
C06147=1101.655,307.498,418.967,179.211,16.906,151.763
C06148=1101.661,307.746,418.936,179.214,16.908,151.763
C06149=1101.667,307.995,418.905,179.218,16.910,151.763
C06150=1101.673,308.242,418.874,179.220,16.911,151.762
C06151=1101.678,308.490,418.843,179.224,16.913,151.762
C06152=1101.684,308.738,418.812,179.227,16.915,151.762
C06153=1101.690,308.986,418.781,179.231,16.917,151.762
C06154=1101.696,309.234,418.750,179.234,16.919,151.762
C06155=1101.701,309.482,418.719,179.238,16.921,151.761
C06156=1101.707,309.730,418.688,179.241,16.923,151.761
C06157=1101.713,309.978,418.657,179.245,16.925,151.761
C06158=1101.718,310.226,418.625,179.248,16.927,151.761
C06159=1101.724,310.474,418.595,179.252,16.929,151.760
C06160=1101.730,310.722,418.563,179.254,16.930,151.760
C06161=1101.736,310.970,418.533,179.258,16.932,151.760
C06162=1101.742,311.218,418.501,179.262,16.934,151.760
C06163=1101.747,311.466,418.470,179.265,16.936,151.759
C06164=1101.753,311.713,418.439,179.268,16.938,151.759
C06165=1101.758,311.962,418.407,179.272,16.940,151.759
C06166=1101.764,312.210,418.376,179.275,16.942,151.759
C06167=1101.770,312.458,418.345,179.279,16.944,151.758
C06168=1101.776,312.706,418.313,179.282,16.946,151.758
C06169=1101.782,312.953,418.282,179.286,16.948,151.758
C06170=1101.787,313.202,418.251,179.288,16.950,151.758
C06171=1101.793,313.449,418.219,179.292,16.951,151.758
C06172=1101.800,313.697,418.188,179.295,16.953,151.757
C06173=1101.805,313.945,418.157,179.299,16.955,151.757
C06174=1101.811,314.194,418.125,179.302,16.958,151.757
C06175=1101.816,314.441,418.093,179.306,16.960,151.757
C06176=1101.822,314.690,418.063,179.309,16.961,151.756
C06177=1101.828,314.937,418.031,179.313,16.963,151.756
C06178=1101.834,315.185,417.999,179.316,16.965,151.756
C06179=1101.840,315.433,417.968,179.319,16.968,151.756
C06180=1101.845,315.681,417.937,179.323,16.970,151.756
C06181=1101.854,316.065,417.887,179.328,16.973,151.755
C06182=1101.862,316.449,417.839,179.333,16.976,151.755
C06183=1101.870,316.834,417.789,179.338,16.979,151.755
C06184=1101.879,317.217,417.740,179.343,16.983,151.755
C06185=1101.884,317.465,417.709,179.346,16.985,151.755
C06186=1101.890,317.713,417.676,179.350,16.987,151.754
C06187=1101.896,317.960,417.645,179.353,16.989,151.754
C06188=1101.901,318.209,417.614,179.356,16.991,151.754
C06189=1101.907,318.457,417.582,179.360,16.993,151.754
C06190=1101.913,318.705,417.550,179.363,16.995,151.754
C06191=1101.918,318.952,417.518,179.366,16.998,151.754
C06192=1101.924,319.201,417.486,179.370,17.000,151.754
C06193=1101.929,319.448,417.454,179.373,17.002,151.753
C06194=1101.935,319.696,417.422,179.376,17.004,151.753
C06195=1101.941,319.944,417.391,179.380,17.006,151.753
C06196=1101.947,320.192,417.359,179.383,17.009,151.753
C06197=1101.952,320.440,417.327,179.386,17.011,151.753
C06198=1101.958,320.688,417.295,179.390,17.013,151.753
C06199=1101.964,320.935,417.263,179.393,17.016,151.753
C06200=1101.969,321.184,417.231,179.396,17.018,151.752
C06201=1101.974,321.431,417.199,179.400,17.020,151.752
C06202=1101.980,321.680,417.167,179.403,17.022,151.752
C06203=1101.986,321.927,417.135,179.406,17.024,151.752
C06204=1101.992,322.175,417.103,179.410,17.026,151.752
C06205=1101.997,322.423,417.072,179.413,17.029,151.752
C06206=1102.003,322.671,417.040,179.416,17.031,151.752
C06207=1102.008,322.918,417.007,179.419,17.033,151.751
C06208=1102.014,323.166,416.975,179.423,17.036,151.751
C06209=1102.020,323.415,416.943,179.426,17.038,151.751
C06210=1102.025,323.662,416.911,179.429,17.040,151.751
C06211=1102.031,323.910,416.879,179.432,17.042,151.751
C06212=1102.037,324.158,416.847,179.436,17.044,151.751
C06213=1102.042,324.406,416.814,179.440,17.047,151.751
C06214=1102.048,324.654,416.782,179.443,17.050,151.751
C06215=1102.054,324.901,416.750,179.447,17.052,151.750
C06216=1102.060,325.150,416.718,179.450,17.054,151.750
C06217=1102.065,325.398,416.685,179.453,17.056,151.750
C06218=1102.070,325.645,416.653,179.456,17.059,151.750
C06219=1102.076,325.893,416.621,179.460,17.061,151.750
C06220=1102.083,326.141,416.589,179.463,17.063,151.750
C06221=1102.088,326.388,416.557,179.466,17.065,151.750
C06222=1102.093,326.637,416.524,179.469,17.068,151.750
C06223=1102.100,326.885,416.492,179.473,17.070,151.750
C06224=1102.105,327.132,416.460,179.476,17.072,151.750
C06225=1102.110,327.381,416.427,179.479,17.075,151.749
C06226=1102.117,327.628,416.394,179.482,17.077,151.749
C06227=1102.123,327.876,416.362,179.486,17.079,151.749
C06228=1102.128,328.123,416.330,179.489,17.082,151.749
C06229=1102.134,328.372,416.297,179.492,17.084,151.749
C06230=1102.140,328.619,416.265,179.496,17.087,151.749
C06231=1102.146,328.868,416.233,179.499,17.089,151.749
C06232=1102.151,329.115,416.200,179.503,17.091,151.749
C06233=1102.160,329.492,416.151,179.507,17.095,151.749
C06234=1102.169,329.869,416.101,179.512,17.099,151.749
C06235=1102.177,330.246,416.052,179.517,17.102,151.748
C06236=1102.186,330.623,416.002,179.523,17.106,151.748
C06237=1102.192,330.871,415.969,179.526,17.109,151.748
C06238=1102.198,331.119,415.937,179.529,17.111,151.748
C06239=1102.204,331.367,415.904,179.532,17.113,151.748
C06240=1102.209,331.614,415.871,179.535,17.116,151.748
C06241=1102.215,331.862,415.839,179.539,17.118,151.748
C06242=1102.221,332.110,415.806,179.542,17.120,151.748
C06243=1102.227,332.357,415.773,179.545,17.123,151.748
C06244=1102.232,332.606,415.741,179.549,17.126,151.748
C06245=1102.239,332.853,415.708,179.552,17.129,151.748
C06246=1102.244,333.101,415.675,179.555,17.131,151.748
C06247=1102.249,333.349,415.642,179.558,17.134,151.748
C06248=1102.255,333.597,415.610,179.562,17.136,151.748
C06249=1102.261,333.845,415.576,179.565,17.138,151.748
C06250=1102.266,334.093,415.543,179.568,17.141,151.748
C06251=1102.272,334.339,415.510,179.572,17.144,151.747
C06252=1102.277,334.588,415.478,179.575,17.146,151.747
C06253=1102.284,334.836,415.445,179.578,17.149,151.747
C06254=1102.289,335.083,415.412,179.581,17.151,151.747
C06255=1102.295,335.331,415.378,179.584,17.154,151.747
C06256=1102.301,335.579,415.346,179.587,17.157,151.748
C06257=1102.306,335.826,415.313,179.591,17.160,151.748
C06258=1102.311,336.074,415.279,179.594,17.162,151.748
C06259=1102.318,336.322,415.247,179.597,17.165,151.747
C06260=1102.323,336.570,415.214,179.600,17.167,151.747
C06261=1102.329,336.818,415.181,179.603,17.170,151.747
C06262=1102.335,337.066,415.148,179.607,17.173,151.747
C06263=1102.340,337.314,415.115,179.610,17.176,151.747
C06264=1102.346,337.562,415.081,179.613,17.178,151.747
C06265=1102.352,337.809,415.048,179.617,17.181,151.747
C06266=1102.357,338.056,415.016,179.619,17.183,151.748
C06267=1102.363,338.304,414.982,179.623,17.187,151.747
C06268=1102.369,338.551,414.948,179.626,17.189,151.747
C06269=1102.375,338.799,414.915,179.630,17.192,151.747
C06270=1102.380,339.047,414.882,179.633,17.194,151.747
C06271=1102.386,339.295,414.849,179.635,17.197,151.748
C06272=1102.392,339.543,414.815,179.639,17.200,151.748
C06273=1102.397,339.791,414.782,179.642,17.203,151.748
C06274=1102.403,340.039,414.749,179.645,17.206,151.748
C06275=1102.408,340.287,414.715,179.648,17.208,151.748
C06276=1102.415,340.534,414.683,179.652,17.212,151.748
C06277=1102.420,340.781,414.649,179.655,17.214,151.748
C06278=1102.426,341.029,414.615,179.658,17.217,151.748
C06279=1102.432,341.277,414.582,179.661,17.220,151.748
C06280=1102.437,341.525,414.549,179.665,17.223,151.748
C06281=1102.442,341.772,414.515,179.668,17.226,151.748
C06282=1102.448,342.020,414.482,179.671,17.228,151.748
C06283=1102.453,342.267,414.448,179.674,17.231,151.748
C06284=1102.459,342.515,414.415,179.678,17.234,151.748
C06285=1102.468,342.886,414.365,179.682,17.238,151.748
C06286=1102.476,343.257,414.314,179.687,17.243,151.748
C06287=1102.485,343.628,414.264,179.692,17.247,151.748
C06288=1102.494,343.998,414.214,179.696,17.251,151.749
C06289=1102.499,344.246,414.181,179.700,17.255,151.749
C06290=1102.506,344.494,414.146,179.703,17.257,151.749
C06291=1102.511,344.742,414.113,179.706,17.260,151.749
C06292=1102.517,344.989,414.079,179.709,17.264,151.749
C06293=1102.523,345.237,414.045,179.713,17.266,151.749
C06294=1102.529,345.485,414.011,179.715,17.269,151.749
C06295=1102.533,345.733,413.977,179.718,17.272,151.749
C06296=1102.539,345.981,413.944,179.722,17.275,151.749
C06297=1102.545,346.228,413.910,179.725,17.278,151.749
C06298=1102.551,346.475,413.876,179.728,17.281,151.749
C06299=1102.556,346.723,413.843,179.731,17.284,151.750
C06300=1102.562,346.970,413.809,179.734,17.287,151.750
C06301=1102.568,347.218,413.775,179.737,17.290,151.750
C06302=1102.574,347.466,413.741,179.741,17.293,151.750
C06303=1102.578,347.714,413.707,179.744,17.296,151.750
C06304=1102.584,347.961,413.673,179.747,17.299,151.750
C06305=1102.590,348.208,413.639,179.750,17.303,151.750
C06306=1102.596,348.457,413.605,179.753,17.306,151.750
C06307=1102.602,348.704,413.571,179.757,17.309,151.751
C06308=1102.607,348.952,413.537,179.759,17.312,151.751
C06309=1102.613,349.200,413.503,179.762,17.315,151.751
C06310=1102.619,349.447,413.469,179.766,17.319,151.751
C06311=1102.625,349.694,413.435,179.769,17.321,151.751
C06312=1102.630,349.942,413.401,179.772,17.324,151.751
C06313=1102.635,350.190,413.367,179.775,17.328,151.751
C06314=1102.642,350.438,413.333,179.778,17.331,151.752
C06315=1102.648,350.685,413.299,179.781,17.334,151.752
C06316=1102.653,350.933,413.264,179.785,17.337,151.752
C06317=1102.659,351.180,413.230,179.787,17.340,151.752
C06318=1102.664,351.428,413.197,179.791,17.344,151.752
C06319=1102.670,351.675,413.163,179.794,17.347,151.752
C06320=1102.676,351.923,413.128,179.796,17.350,151.753
C06321=1102.682,352.171,413.094,179.800,17.353,151.753
C06322=1102.687,352.418,413.060,179.803,17.356,151.753
C06323=1102.693,352.666,413.025,179.806,17.360,151.753
C06324=1102.698,352.913,412.991,179.809,17.363,151.753
C06325=1102.705,353.161,412.957,179.812,17.366,151.753
C06326=1102.710,353.408,412.922,179.815,17.370,151.754
C06327=1102.716,353.656,412.888,179.818,17.373,151.754
C06328=1102.722,353.903,412.854,179.822,17.377,151.754
C06329=1102.727,354.151,412.819,179.824,17.379,151.754
C06330=1102.733,354.399,412.785,179.828,17.383,151.754
C06331=1102.738,354.646,412.750,179.831,17.386,151.755
C06332=1102.744,354.894,412.716,179.833,17.389,151.755
C06333=1102.749,355.141,412.681,179.837,17.393,151.755
C06334=1102.756,355.389,412.647,179.840,17.396,151.755
C06335=1102.761,355.637,412.612,179.843,17.400,151.756
C06336=1102.767,355.884,412.578,179.846,17.403,151.756
C06337=1102.775,356.257,412.526,179.850,17.409,151.756
C06338=1102.784,356.630,412.474,179.855,17.414,151.756
C06339=1102.792,357.003,412.421,179.859,17.418,151.757
C06340=1102.801,357.376,412.370,179.864,17.424,151.757
C06341=1102.806,357.623,412.335,179.868,17.427,151.757
C06342=1102.813,357.871,412.300,179.870,17.431,151.758
C06343=1102.818,358.119,412.266,179.874,17.435,151.758
C06344=1102.824,358.366,412.231,179.876,17.438,151.758
C06345=1102.830,358.614,412.196,179.880,17.442,151.758
C06346=1102.836,358.861,412.162,179.882,17.445,151.759
C06347=1102.841,359.109,412.127,179.886,17.449,151.759
C06348=1102.847,359.356,412.091,179.888,17.452,151.759
C06349=1102.853,359.604,412.057,179.892,17.456,151.759
C06350=1102.858,359.851,412.023,179.894,17.459,151.760
C06351=1102.864,360.099,411.987,179.898,17.463,151.760
C06352=1102.870,360.346,411.953,179.900,17.466,151.760
C06353=1102.875,360.593,411.917,179.904,17.470,151.761
C06354=1102.882,360.841,411.883,179.906,17.473,151.761
C06355=1102.887,361.089,411.848,179.910,17.477,151.761
C06356=1102.892,361.336,411.813,179.912,17.480,151.761
C06357=1102.898,361.584,411.778,179.916,17.484,151.762
C06358=1102.904,361.831,411.743,179.918,17.488,151.762
C06359=1102.909,362.078,411.709,179.922,17.492,151.762
C06360=1102.915,362.326,411.673,179.924,17.495,151.763
C06361=1102.920,362.574,411.638,179.927,17.499,151.763
C06362=1102.927,362.821,411.603,179.931,17.503,151.763
C06363=1102.932,363.068,411.568,179.933,17.506,151.764
C06364=1102.938,363.316,411.533,179.936,17.510,151.764
C06365=1102.944,363.563,411.497,179.939,17.514,151.764
C06366=1102.949,363.811,411.463,179.942,17.518,151.765
C06367=1102.955,364.058,411.428,179.945,17.521,151.765
C06368=1102.961,364.305,411.392,179.948,17.525,151.765
C06369=1102.966,364.553,411.358,179.951,17.529,151.766
C06370=1102.972,364.800,411.322,179.954,17.533,151.766
C06371=1102.978,365.047,411.287,179.957,17.537,151.766
C06372=1102.984,365.295,411.252,179.960,17.540,151.767
C06373=1102.989,365.542,411.217,179.963,17.544,151.767
C06374=1102.995,365.790,411.181,179.966,17.548,151.767
C06375=1103.001,366.037,411.146,179.969,17.552,151.768
C06376=1103.007,366.285,411.111,179.972,17.556,151.768
C06377=1103.012,366.532,411.075,179.974,17.560,151.769
C06378=1103.017,366.779,411.040,179.978,17.563,151.769
C06379=1103.023,367.027,411.004,179.981,17.568,151.769
C06380=1103.029,367.274,410.969,179.983,17.572,151.770
C06381=1103.035,367.522,410.933,179.986,17.575,151.770
C06382=1103.040,367.769,410.898,179.989,17.579,151.771
C06383=1103.046,368.017,410.863,179.992,17.583,151.771
C06384=1103.051,368.264,410.827,179.995,17.587,151.771
C06385=1103.058,368.512,410.792,179.997,17.591,151.772
C06386=1103.063,368.758,410.756,-180.000,17.595,151.772
C06387=1103.068,369.005,410.721,-179.996,17.599,151.773
C06388=1103.074,369.253,410.685,-179.994,17.603,151.773
C06389=1103.082,369.591,410.637,-179.990,17.609,151.774
C06390=1103.090,369.930,410.588,-179.986,17.615,151.774
C06391=1103.098,370.268,410.539,-179.982,17.620,151.775
C06392=1103.106,370.607,410.490,-179.978,17.626,151.776
C06393=1103.112,370.854,410.455,-179.975,17.630,151.776
C06394=1103.118,371.101,410.419,-179.973,17.634,151.776
C06395=1103.123,371.348,410.384,-179.969,17.638,151.777
C06396=1103.128,371.596,410.347,-179.966,17.642,151.777
C06397=1103.134,371.843,410.312,-179.964,17.646,151.778
C06398=1103.140,372.091,410.276,-179.961,17.650,151.778
C06399=1103.145,372.338,410.241,-179.958,17.655,151.779
C06400=1103.152,372.585,410.204,-179.956,17.658,151.779
C06401=1103.158,372.833,410.169,-179.953,17.663,151.780
C06402=1103.163,373.080,410.133,-179.949,17.667,151.780
C06403=1103.169,373.327,410.097,-179.947,17.672,151.781
C06404=1103.174,373.574,410.061,-179.944,17.675,151.781
C06405=1103.180,373.822,410.025,-179.941,17.680,151.782
C06406=1103.186,374.069,409.989,-179.938,17.684,151.782
C06407=1103.192,374.316,409.954,-179.935,17.688,151.782
C06408=1103.198,374.563,409.918,-179.933,17.693,151.783
C06409=1103.203,374.811,409.881,-179.930,17.697,151.784
C06410=1103.209,375.058,409.846,-179.927,17.701,151.784
C06411=1103.215,375.305,409.809,-179.924,17.706,151.785
C06412=1103.220,375.553,409.773,-179.922,17.710,151.785
C06413=1103.226,375.800,409.738,-179.919,17.714,151.786
C06414=1103.231,376.047,409.702,-179.916,17.719,151.786
C06415=1103.237,376.295,409.665,-179.913,17.723,151.787
C06416=1103.243,376.542,409.629,-179.911,17.727,151.787
C06417=1103.248,376.789,409.593,-179.908,17.732,151.788
C06418=1103.254,377.036,409.556,-179.905,17.737,151.789
C06419=1103.260,377.284,409.521,-179.902,17.741,151.789
C06420=1103.265,377.530,409.484,-179.899,17.746,151.790
C06421=1103.271,377.778,409.448,-179.897,17.750,151.790
C06422=1103.277,378.025,409.412,-179.894,17.754,151.791
C06423=1103.282,378.272,409.376,-179.891,17.759,151.791
C06424=1103.288,378.519,409.339,-179.889,17.764,151.792
C06425=1103.295,378.816,409.296,-179.885,17.769,151.793
C06426=1103.302,379.113,409.253,-179.882,17.774,151.793
C06427=1103.309,379.410,409.209,-179.879,17.780,151.794
C06428=1103.315,379.707,409.165,-179.876,17.785,151.795
C06429=1103.321,379.954,409.129,-179.873,17.790,151.795
C06430=1103.328,380.201,409.092,-179.870,17.795,151.796
C06431=1103.332,380.448,409.056,-179.867,17.799,151.797
C06432=1103.339,380.695,409.020,-179.865,17.803,151.797
C06433=1103.344,380.943,408.983,-179.862,17.808,151.798
C06434=1103.350,381.189,408.947,-179.859,17.813,151.798
C06435=1103.355,381.437,408.910,-179.857,17.818,151.799
C06436=1103.362,381.684,408.874,-179.854,17.822,151.800
C06437=1103.367,381.931,408.837,-179.851,17.827,151.800
C06438=1103.374,382.178,408.800,-179.848,17.832,151.801
C06439=1103.378,382.426,408.764,-179.846,17.836,151.802
C06440=1103.385,382.673,408.728,-179.844,17.841,151.802
C06441=1103.394,383.088,408.666,-179.838,17.850,151.803
C06442=1103.404,383.502,408.604,-179.834,17.858,151.805
C06443=1103.413,383.918,408.543,-179.830,17.866,151.806
C06444=1103.422,384.332,408.481,-179.826,17.874,151.807
C06445=1103.429,384.579,408.445,-179.823,17.878,151.808
C06446=1103.434,384.826,408.408,-179.820,17.884,151.808
C06447=1103.440,385.074,408.371,-179.818,17.889,151.809
C06448=1103.445,385.320,408.334,-179.815,17.893,151.810
C06449=1103.451,385.567,408.297,-179.813,17.899,151.810
C06450=1103.457,385.815,408.260,-179.810,17.904,151.811
C06451=1103.462,386.062,408.223,-179.807,17.908,151.812
C06452=1103.468,386.310,408.186,-179.805,17.913,151.813
C06453=1103.474,386.556,408.150,-179.802,17.919,151.813
C06454=1103.479,386.803,408.113,-179.799,17.924,151.814
C06455=1103.485,387.050,408.075,-179.797,17.929,151.815
C06456=1103.491,387.297,408.038,-179.794,17.934,151.816
C06457=1103.497,387.544,408.002,-179.791,17.939,151.816
C06458=1103.503,387.792,407.965,-179.789,17.944,151.817
C06459=1103.508,388.038,407.928,-179.786,17.949,151.818
C06460=1103.514,388.285,407.890,-179.784,17.954,151.819
C06461=1103.519,388.533,407.853,-179.781,17.959,151.819
C06462=1103.525,388.780,407.816,-179.779,17.964,151.820
C06463=1103.531,389.027,407.780,-179.776,17.970,151.821
C06464=1103.537,389.274,407.742,-179.774,17.975,151.822
C06465=1103.543,389.521,407.705,-179.771,17.980,151.823
C06466=1103.548,389.768,407.668,-179.769,17.985,151.823
C06467=1103.554,390.015,407.630,-179.766,17.990,151.824
C06468=1103.560,390.263,407.593,-179.764,17.995,151.825
C06469=1103.565,390.510,407.556,-179.761,18.001,151.826
C06470=1103.572,390.756,407.519,-179.758,18.007,151.827
C06471=1103.577,391.003,407.482,-179.755,18.012,151.827
C06472=1103.583,391.251,407.445,-179.753,18.017,151.828
C06473=1103.588,391.497,407.408,-179.750,18.022,151.829
C06474=1103.594,391.745,407.371,-179.748,18.028,151.830
C06475=1103.600,391.991,407.333,-179.746,18.033,151.831
C06476=1103.606,392.239,407.295,-179.743,18.039,151.832
C06477=1103.612,392.486,407.258,-179.741,18.044,151.833
C06478=1103.618,392.733,407.221,-179.738,18.049,151.833
C06479=1103.623,392.979,407.183,-179.736,18.055,151.834
C06480=1103.629,393.228,407.146,-179.733,18.060,151.835
C06481=1103.635,393.474,407.108,-179.731,18.065,151.836
C06482=1103.641,393.722,407.071,-179.728,18.071,151.837
C06483=1103.647,393.968,407.033,-179.726,18.077,151.838
C06484=1103.651,394.216,406.996,-179.723,18.082,151.839
C06485=1103.657,394.463,406.958,-179.721,18.088,151.840
C06486=1103.663,394.710,406.920,-179.719,18.093,151.841
C06487=1103.669,394.957,406.883,-179.716,18.099,151.842
C06488=1103.675,395.204,406.845,-179.714,18.104,151.843
C06489=1103.681,395.450,406.808,-179.712,18.110,151.843
C06490=1103.686,395.698,406.771,-179.709,18.116,151.844
C06491=1103.691,395.945,406.732,-179.706,18.122,151.845
C06492=1103.697,396.192,406.694,-179.704,18.127,151.846
C06493=1103.702,396.405,406.662,-179.703,18.132,151.847
C06494=1103.707,396.619,406.630,-179.700,18.137,151.848
C06495=1103.713,396.833,406.597,-179.698,18.142,151.849
C06496=1103.717,397.046,406.564,-179.696,18.147,151.850
C06497=1103.722,397.260,406.531,-179.694,18.152,151.851
C06498=1103.727,397.473,406.499,-179.692,18.157,151.851
C06499=1103.732,397.686,406.466,-179.690,18.162,151.852
C06500=1103.737,397.899,406.434,-179.688,18.167,151.853
C06501=1103.743,398.147,406.395,-179.685,18.173,151.854
C06502=1103.748,398.395,406.358,-179.683,18.178,151.855
C06503=1103.754,398.641,406.320,-179.680,18.185,151.856
C06504=1103.759,398.888,406.282,-179.678,18.191,151.857
C06505=1103.765,399.135,406.244,-179.676,18.196,151.858
C06506=1103.771,399.382,406.206,-179.674,18.202,151.859
C06507=1103.777,399.630,406.168,-179.671,18.209,151.860
C06508=1103.783,399.876,406.130,-179.669,18.215,151.861
C06509=1103.789,400.123,406.092,-179.667,18.220,151.862
C06510=1103.794,400.370,406.054,-179.665,18.226,151.863
C06511=1103.800,400.617,406.016,-179.662,18.233,151.864
C06512=1103.805,400.864,405.978,-179.660,18.238,151.865
C06513=1103.812,401.111,405.940,-179.657,18.244,151.867
C06514=1103.817,401.359,405.901,-179.655,18.251,151.868
C06515=1103.823,401.605,405.863,-179.653,18.257,151.869
C06516=1103.828,401.852,405.825,-179.651,18.263,151.870
C06517=1103.834,402.100,405.787,-179.648,18.269,151.871
C06518=1103.840,402.347,405.749,-179.646,18.275,151.872
C06519=1103.845,402.594,405.711,-179.644,18.282,151.873
C06520=1103.852,402.840,405.672,-179.641,18.288,151.874
C06521=1103.857,403.087,405.634,-179.639,18.294,151.875
C06522=1103.863,403.334,405.595,-179.637,18.300,151.877
C06523=1103.868,403.581,405.558,-179.634,18.307,151.878
C06524=1103.874,403.828,405.519,-179.633,18.313,151.879
C06525=1103.880,404.075,405.480,-179.630,18.319,151.880
C06526=1103.886,404.322,405.442,-179.628,18.326,151.881
C06527=1103.892,404.569,405.404,-179.626,18.332,151.882
C06528=1103.897,404.817,405.366,-179.623,18.339,151.884
C06529=1103.903,405.063,405.327,-179.621,18.345,151.885
C06530=1103.909,405.310,405.289,-179.618,18.351,151.886
C06531=1103.914,405.558,405.250,-179.617,18.358,151.887
C06532=1103.921,405.804,405.212,-179.615,18.364,151.888
C06533=1103.926,406.051,405.173,-179.612,18.371,151.890
C06534=1103.932,406.299,405.135,-179.610,18.377,151.891
C06535=1103.938,406.545,405.096,-179.608,18.384,151.892
C06536=1103.943,406.792,405.058,-179.606,18.390,151.893
C06537=1103.949,407.039,405.018,-179.603,18.397,151.894
C06538=1103.954,407.286,404.980,-179.601,18.404,151.896
C06539=1103.960,407.533,404.942,-179.599,18.411,151.897
C06540=1103.966,407.780,404.903,-179.597,18.417,151.898
C06541=1103.971,408.027,404.864,-179.594,18.424,151.899
C06542=1103.977,408.273,404.825,-179.593,18.430,151.901
C06543=1103.983,408.521,404.787,-179.590,18.438,151.902
C06544=1103.989,408.767,404.748,-179.588,18.444,151.903
C06545=1103.994,409.014,404.709,-179.586,18.451,151.905
C06546=1104.000,409.261,404.670,-179.584,18.458,151.906
C06547=1104.005,409.508,404.631,-179.582,18.465,151.907
C06548=1104.011,409.756,404.593,-179.579,18.472,151.909
C06549=1104.016,409.969,404.559,-179.577,18.478,151.910
C06550=1104.021,410.182,404.525,-179.576,18.483,151.911
C06551=1104.026,410.395,404.492,-179.574,18.490,151.912
C06552=1104.031,410.608,404.458,-179.572,18.496,151.913
C06553=1104.036,410.822,404.424,-179.570,18.502,151.914
C06554=1104.041,411.036,404.391,-179.569,18.508,151.916
C06555=1104.046,411.249,404.357,-179.566,18.514,151.917
C06556=1104.051,411.462,404.323,-179.565,18.520,151.918
C06557=1104.056,411.710,404.284,-179.563,18.527,151.919
C06558=1104.062,411.956,404.245,-179.561,18.534,151.921
C06559=1104.068,412.203,404.206,-179.558,18.541,151.922
C06560=1104.073,412.450,404.167,-179.557,18.549,151.924
C06561=1104.079,412.697,404.127,-179.554,18.556,151.925
C06562=1104.085,412.944,404.089,-179.552,18.563,151.926
C06563=1104.091,413.191,404.050,-179.550,18.570,151.928
C06564=1104.096,413.438,404.011,-179.548,18.577,151.929
C06565=1104.102,413.685,403.971,-179.546,18.585,151.931
C06566=1104.108,413.931,403.932,-179.544,18.592,151.932
C06567=1104.114,414.178,403.893,-179.542,18.599,151.934
C06568=1104.119,414.425,403.854,-179.540,18.607,151.935
C06569=1104.125,414.672,403.814,-179.537,18.614,151.936
C06570=1104.131,414.918,403.775,-179.536,18.621,151.938
C06571=1104.137,415.165,403.736,-179.534,18.629,151.939
C06572=1104.142,415.412,403.697,-179.532,18.636,151.941
C06573=1104.148,415.659,403.657,-179.529,18.644,151.942
C06574=1104.155,415.906,403.618,-179.527,18.651,151.944
C06575=1104.160,416.153,403.579,-179.526,18.658,151.945
C06576=1104.166,416.400,403.539,-179.524,18.666,151.947
C06577=1104.172,416.646,403.500,-179.521,18.674,151.948
C06578=1104.178,416.893,403.460,-179.519,18.681,151.950
C06579=1104.183,417.139,403.421,-179.517,18.689,151.951
C06580=1104.189,417.387,403.381,-179.515,18.697,151.953
C06581=1104.195,417.634,403.342,-179.514,18.704,151.955
C06582=1104.200,417.880,403.302,-179.512,18.712,151.956
C06583=1104.207,418.127,403.262,-179.510,18.720,151.958
C06584=1104.211,418.373,403.223,-179.508,18.727,151.959
C06585=1104.217,418.621,403.183,-179.506,18.735,151.961
C06586=1104.223,418.867,403.144,-179.504,18.743,151.963
C06587=1104.229,419.113,403.104,-179.501,18.751,151.964
C06588=1104.235,419.361,403.064,-179.500,18.759,151.966
C06589=1104.240,419.607,403.025,-179.498,18.767,151.968
C06590=1104.246,419.854,402.985,-179.496,18.775,151.969
C06591=1104.251,420.101,402.945,-179.495,18.783,151.971
C06592=1104.257,420.348,402.906,-179.493,18.791,151.973
C06593=1104.264,420.594,402.866,-179.491,18.799,151.974
C06594=1104.268,420.841,402.826,-179.489,18.807,151.976
C06595=1104.275,421.088,402.786,-179.487,18.815,151.977
C06596=1104.281,421.335,402.746,-179.485,18.823,151.979
C06597=1104.286,421.581,402.706,-179.483,18.831,151.981
C06598=1104.292,421.828,402.666,-179.481,18.839,151.982
C06599=1104.298,422.074,402.626,-179.479,18.847,151.984
C06600=1104.304,422.322,402.586,-179.477,18.855,151.986
C06601=1104.309,422.568,402.547,-179.475,18.864,151.988
C06602=1104.315,422.815,402.506,-179.474,18.872,151.989
C06603=1104.321,423.062,402.466,-179.472,18.880,151.991
C06604=1104.327,423.307,402.427,-179.469,18.889,151.993
C06605=1104.332,423.528,402.391,-179.468,18.896,151.995
C06606=1104.337,423.748,402.355,-179.467,18.904,151.996
C06607=1104.342,423.969,402.319,-179.464,18.911,151.998
C06608=1104.347,424.189,402.283,-179.463,18.919,151.999
C06609=1104.352,424.408,402.247,-179.461,18.927,152.001
C06610=1104.357,424.629,402.212,-179.460,18.934,152.003
C06611=1104.362,424.849,402.176,-179.458,18.942,152.004
C06612=1104.367,425.069,402.140,-179.457,18.949,152.006
C06613=1104.374,425.316,402.100,-179.455,18.958,152.008
C06614=1104.379,425.562,402.059,-179.453,18.966,152.010
C06615=1104.384,425.809,402.019,-179.452,18.975,152.012
C06616=1104.391,426.055,401.979,-179.449,18.984,152.013
C06617=1104.396,426.302,401.938,-179.448,18.993,152.015
C06618=1104.402,426.549,401.898,-179.446,19.002,152.017
C06619=1104.407,426.795,401.858,-179.445,19.010,152.019
C06620=1104.413,427.042,401.817,-179.443,19.019,152.021
C06621=1104.419,427.288,401.777,-179.441,19.028,152.023
C06622=1104.425,427.535,401.736,-179.439,19.037,152.025
C06623=1104.430,427.781,401.696,-179.438,19.046,152.027
C06624=1104.436,428.028,401.656,-179.436,19.055,152.029
C06625=1104.442,428.275,401.615,-179.435,19.063,152.031
C06626=1104.448,428.521,401.575,-179.432,19.073,152.033
C06627=1104.454,428.768,401.534,-179.431,19.082,152.035
C06628=1104.460,429.015,401.493,-179.429,19.090,152.037
C06629=1104.465,429.261,401.453,-179.428,19.100,152.039
C06630=1104.471,429.507,401.412,-179.426,19.109,152.041
C06631=1104.477,429.754,401.371,-179.424,19.118,152.043
C06632=1104.483,430.001,401.331,-179.423,19.127,152.045
C06633=1104.488,430.247,401.290,-179.421,19.137,152.047
C06634=1104.493,430.494,401.250,-179.419,19.146,152.049
C06635=1104.500,430.740,401.209,-179.418,19.155,152.051
C06636=1104.506,430.986,401.168,-179.417,19.164,152.053
C06637=1104.511,431.233,401.127,-179.415,19.174,152.055
C06638=1104.517,431.480,401.087,-179.413,19.183,152.057
C06639=1104.523,431.726,401.045,-179.411,19.193,152.059
C06640=1104.529,431.973,401.004,-179.410,19.202,152.061
C06641=1104.534,432.220,400.964,-179.409,19.211,152.063
C06642=1104.540,432.465,400.923,-179.407,19.222,152.066
C06643=1104.546,432.712,400.882,-179.405,19.231,152.068
C06644=1104.552,432.959,400.842,-179.404,19.240,152.070
C06645=1104.558,433.205,400.800,-179.402,19.250,152.072
C06646=1104.563,433.452,400.759,-179.401,19.260,152.074
C06647=1104.569,433.698,400.718,-179.399,19.270,152.076
C06648=1104.575,433.945,400.677,-179.398,19.279,152.079
C06649=1104.581,434.191,400.636,-179.396,19.289,152.081
C06650=1104.586,434.438,400.595,-179.395,19.299,152.083
C06651=1104.592,434.684,400.554,-179.394,19.309,152.086
C06652=1104.597,434.930,400.513,-179.392,19.319,152.088
C06653=1104.603,435.176,400.472,-179.391,19.329,152.090
C06654=1104.609,435.423,400.431,-179.389,19.339,152.092
C06655=1104.614,435.670,400.389,-179.388,19.349,152.095
C06656=1104.620,435.916,400.348,-179.387,19.359,152.097
C06657=1104.626,436.163,400.307,-179.386,19.369,152.099
C06658=1104.632,436.409,400.265,-179.384,19.379,152.102
C06659=1104.638,436.655,400.224,-179.383,19.389,152.104
C06660=1104.643,436.902,400.183,-179.381,19.399,152.106
C06661=1104.653,437.320,400.113,-179.379,19.417,152.110
C06662=1104.658,437.528,400.077,-179.377,19.426,152.112
C06663=1104.663,437.736,400.042,-179.377,19.434,152.114
C06664=1104.668,437.946,400.008,-179.375,19.443,152.116
C06665=1104.673,438.154,399.972,-179.375,19.452,152.118
C06666=1104.677,438.363,399.938,-179.373,19.461,152.120
C06667=1104.683,438.572,399.903,-179.373,19.469,152.123
C06668=1104.688,438.818,399.860,-179.371,19.480,152.125
C06669=1104.694,439.064,399.819,-179.369,19.491,152.127
C06670=1104.700,439.311,399.778,-179.369,19.501,152.130
C06671=1104.706,439.557,399.736,-179.367,19.512,152.132
C06672=1104.712,439.803,399.695,-179.365,19.523,152.135
C06673=1104.717,440.049,399.653,-179.365,19.533,152.137
C06674=1104.723,440.296,399.611,-179.363,19.544,152.140
C06675=1104.729,440.542,399.570,-179.363,19.554,152.142
C06676=1104.735,440.788,399.528,-179.361,19.566,152.145
C06677=1104.740,441.035,399.486,-179.360,19.577,152.148
C06678=1104.747,441.282,399.444,-179.358,19.588,152.150
C06679=1104.752,441.528,399.402,-179.358,19.598,152.153
C06680=1104.758,441.774,399.361,-179.357,19.610,152.155
C06681=1104.764,442.020,399.319,-179.355,19.621,152.158
C06682=1104.769,442.267,399.277,-179.355,19.631,152.161
C06683=1104.775,442.513,399.236,-179.353,19.643,152.163
C06684=1104.781,442.759,399.194,-179.352,19.654,152.166
C06685=1104.786,443.005,399.152,-179.351,19.665,152.168
C06686=1104.792,443.251,399.110,-179.350,19.676,152.171
C06687=1104.797,443.498,399.068,-179.349,19.688,152.174
C06688=1104.804,443.744,399.026,-179.348,19.699,152.177
C06689=1104.810,443.991,398.984,-179.347,19.710,152.179
C06690=1104.815,444.237,398.942,-179.347,19.721,152.182
C06691=1104.821,444.483,398.899,-179.346,19.733,152.185
C06692=1104.827,444.729,398.858,-179.346,19.744,152.188
C06693=1104.832,444.976,398.816,-179.346,19.755,152.191
C06694=1104.839,445.222,398.773,-179.345,19.767,152.193
C06695=1104.844,445.468,398.731,-179.346,19.777,152.196
C06696=1104.849,445.715,398.689,-179.346,19.789,152.199
C06697=1104.856,445.960,398.647,-179.347,19.800,152.202
C06698=1104.861,446.207,398.605,-179.346,19.811,152.205
C06699=1104.868,446.453,398.562,-179.347,19.822,152.208
C06700=1104.873,446.700,398.520,-179.348,19.833,152.211
C06701=1104.878,446.946,398.478,-179.349,19.844,152.214
C06702=1104.884,447.192,398.436,-179.350,19.855,152.217
C06703=1104.890,447.438,398.393,-179.351,19.866,152.220
C06704=1104.896,447.685,398.351,-179.351,19.877,152.223
C06705=1104.901,447.931,398.308,-179.353,19.888,152.226
C06706=1104.907,448.177,398.267,-179.354,19.899,152.229
C06707=1104.913,448.423,398.224,-179.356,19.910,152.232
C06708=1104.919,448.670,398.182,-179.357,19.922,152.235
C06709=1104.925,448.916,398.139,-179.358,19.932,152.238
C06710=1104.930,449.162,398.097,-179.360,19.943,152.241
C06711=1104.936,449.409,398.054,-179.362,19.954,152.244
C06712=1104.941,449.655,398.012,-179.364,19.965,152.247
C06713=1104.948,449.901,397.970,-179.366,19.976,152.250
C06714=1104.953,450.147,397.927,-179.367,19.987,152.254
C06715=1104.959,450.394,397.885,-179.369,19.998,152.257
C06716=1104.555,450.386,397.757,-179.445,20.226,152.328
C06717=1104.549,450.140,397.800,-179.443,20.215,152.325
C06718=1104.544,449.893,397.842,-179.441,20.204,152.322
C06719=1104.537,449.647,397.885,-179.440,20.193,152.319
C06720=1104.532,449.401,397.927,-179.438,20.182,152.316
C06721=1104.526,449.154,397.970,-179.436,20.171,152.312
C06722=1104.520,448.908,398.012,-179.434,20.160,152.309
C06723=1104.514,448.663,398.055,-179.433,20.150,152.306
C06724=1104.509,448.416,398.097,-179.432,20.138,152.303
C06725=1104.503,448.170,398.140,-179.430,20.127,152.300
C06726=1104.498,447.923,398.182,-179.429,20.116,152.297
C06727=1104.491,447.678,398.224,-179.428,20.105,152.294
C06728=1104.485,447.431,398.267,-179.427,20.094,152.291
C06729=1104.480,447.184,398.309,-179.426,20.082,152.288
C06730=1104.475,446.939,398.352,-179.425,20.071,152.285
C06731=1104.469,446.692,398.393,-179.424,20.060,152.282
C06732=1104.463,446.446,398.437,-179.424,20.049,152.279
C06733=1104.457,446.199,398.479,-179.423,20.038,152.276
C06734=1104.451,445.954,398.521,-179.423,20.026,152.273
C06735=1104.446,445.707,398.563,-179.422,20.015,152.270
C06736=1104.439,445.461,398.605,-179.423,20.004,152.267
C06737=1104.434,445.214,398.647,-179.423,19.992,152.265
C06738=1104.429,444.968,398.690,-179.422,19.982,152.262
C06739=1104.422,444.722,398.732,-179.423,19.970,152.259
C06740=1104.417,444.476,398.774,-179.423,19.959,152.256
C06741=1104.410,444.229,398.816,-179.424,19.947,152.253
C06742=1104.405,443.983,398.858,-179.424,19.936,152.250
C06743=1104.399,443.737,398.900,-179.425,19.925,152.248
C06744=1104.394,443.491,398.943,-179.426,19.914,152.245
C06745=1104.388,443.245,398.984,-179.427,19.902,152.242
C06746=1104.382,442.998,399.026,-179.429,19.890,152.240
C06747=1104.376,442.752,399.069,-179.429,19.880,152.237
C06748=1104.370,442.505,399.111,-179.431,19.868,152.234
C06749=1104.364,442.259,399.152,-179.432,19.857,152.232
C06750=1104.359,442.013,399.194,-179.433,19.846,152.229
C06751=1104.353,441.767,399.236,-179.434,19.835,152.226
C06752=1104.347,441.521,399.278,-179.435,19.824,152.224
C06753=1104.342,441.274,399.320,-179.437,19.812,152.221
C06754=1104.336,441.028,399.361,-179.437,19.802,152.218
C06755=1104.330,440.782,399.403,-179.439,19.791,152.216
C06756=1104.325,440.535,399.445,-179.440,19.779,152.213
C06757=1104.318,440.289,399.487,-179.442,19.768,152.211
C06758=1104.312,440.042,399.528,-179.443,19.758,152.208
C06759=1104.307,439.796,399.570,-179.444,19.747,152.206
C06760=1104.301,439.550,399.612,-179.445,19.736,152.203
C06761=1104.295,439.303,399.653,-179.446,19.726,152.201
C06762=1104.289,439.057,399.695,-179.448,19.715,152.198
C06763=1104.283,438.811,399.736,-179.449,19.705,152.196
C06764=1104.278,438.564,399.778,-179.451,19.694,152.193
C06765=1104.268,438.152,399.847,-179.453,19.676,152.189
C06766=1104.258,437.740,399.917,-179.455,19.659,152.185
C06767=1104.249,437.328,399.986,-179.457,19.641,152.181
C06768=1104.239,436.915,400.056,-179.460,19.624,152.177
C06769=1104.233,436.669,400.097,-179.462,19.613,152.175
C06770=1104.227,436.422,400.138,-179.462,19.603,152.172
C06771=1104.221,436.176,400.180,-179.464,19.593,152.170
C06772=1104.215,435.930,400.221,-179.465,19.583,152.168
C06773=1104.209,435.684,400.262,-179.467,19.573,152.166
C06774=1104.204,435.437,400.304,-179.468,19.563,152.163
C06775=1104.199,435.190,400.345,-179.470,19.552,152.161
C06776=1104.193,434.944,400.387,-179.471,19.543,152.159
C06777=1104.187,434.697,400.427,-179.473,19.532,152.156
C06778=1104.181,434.451,400.469,-179.474,19.522,152.154
C06779=1104.176,434.205,400.509,-179.476,19.512,152.152
C06780=1104.170,433.959,400.551,-179.477,19.502,152.149
C06781=1104.164,433.712,400.591,-179.478,19.493,152.147
C06782=1104.158,433.466,400.633,-179.480,19.483,152.145
C06783=1104.153,433.219,400.674,-179.481,19.473,152.143
C06784=1104.147,432.973,400.715,-179.484,19.463,152.141
C06785=1104.141,432.726,400.756,-179.485,19.454,152.138
C06786=1104.135,432.480,400.797,-179.487,19.444,152.136
C06787=1104.130,432.233,400.838,-179.488,19.434,152.134
C06788=1104.124,431.987,400.880,-179.489,19.425,152.132
C06789=1104.118,431.740,400.920,-179.492,19.415,152.130
C06790=1104.112,431.493,400.960,-179.493,19.406,152.128
C06791=1104.106,431.248,401.001,-179.494,19.396,152.126
C06792=1104.101,431.001,401.042,-179.496,19.387,152.124
C06793=1104.095,430.754,401.083,-179.498,19.377,152.121
C06794=1104.089,430.507,401.124,-179.499,19.368,152.119
C06795=1104.083,430.261,401.165,-179.501,19.358,152.117
C06796=1104.078,430.014,401.206,-179.503,19.349,152.115
C06797=1104.071,429.768,401.246,-179.504,19.340,152.113
C06798=1104.066,429.522,401.286,-179.506,19.330,152.111
C06799=1104.061,429.275,401.327,-179.508,19.321,152.109
C06800=1104.055,429.029,401.369,-179.509,19.312,152.107
C06801=1104.048,428.782,401.409,-179.511,19.303,152.105
C06802=1104.043,428.535,401.450,-179.513,19.294,152.103
C06803=1104.037,428.289,401.490,-179.514,19.285,152.101
C06804=1104.031,428.043,401.530,-179.516,19.276,152.099
C06805=1104.026,427.796,401.571,-179.518,19.267,152.097
C06806=1104.020,427.549,401.612,-179.520,19.258,152.095
C06807=1104.014,427.303,401.652,-179.521,19.249,152.093
C06808=1104.008,427.056,401.692,-179.523,19.240,152.091
C06809=1104.002,426.809,401.733,-179.525,19.232,152.089
C06810=1103.997,426.563,401.773,-179.527,19.222,152.088
C06811=1103.991,426.316,401.814,-179.529,19.213,152.086
C06812=1103.985,426.070,401.854,-179.530,19.205,152.084
C06813=1103.979,425.823,401.895,-179.532,19.196,152.082
C06814=1103.974,425.577,401.935,-179.534,19.187,152.080
C06815=1103.968,425.330,401.974,-179.535,19.179,152.078
C06816=1103.962,425.083,402.015,-179.538,19.170,152.076
C06817=1103.957,424.863,402.051,-179.539,19.162,152.075
C06818=1103.952,424.642,402.087,-179.541,19.154,152.073
C06819=1103.947,424.422,402.123,-179.542,19.147,152.071
C06820=1103.942,424.202,402.159,-179.544,19.139,152.070
C06821=1103.937,423.981,402.195,-179.546,19.131,152.068
C06822=1103.932,423.761,402.230,-179.547,19.124,152.066
C06823=1103.927,423.541,402.266,-179.549,19.116,152.065
C06824=1103.921,423.321,402.302,-179.550,19.109,152.063
C06825=1103.916,423.074,402.343,-179.552,19.100,152.061
C06826=1103.909,422.827,402.383,-179.554,19.092,152.060
C06827=1103.904,422.580,402.423,-179.556,19.084,152.058
C06828=1103.898,422.334,402.463,-179.558,19.075,152.056
C06829=1103.892,422.088,402.503,-179.561,19.067,152.054
C06830=1103.887,421.840,402.543,-179.562,19.058,152.053
C06831=1103.881,421.594,402.583,-179.564,19.050,152.051
C06832=1103.875,421.347,402.622,-179.566,19.042,152.049
C06833=1103.869,421.100,402.663,-179.568,19.034,152.047
C06834=1103.864,420.854,402.702,-179.570,19.025,152.046
C06835=1103.858,420.607,402.743,-179.572,19.017,152.044
C06836=1103.852,420.360,402.782,-179.573,19.010,152.042
C06837=1103.846,420.114,402.822,-179.575,19.002,152.041
C06838=1103.841,419.867,402.862,-179.577,18.994,152.039
C06839=1103.835,419.619,402.901,-179.579,18.986,152.037
C06840=1103.829,419.374,402.941,-179.581,18.978,152.036
C06841=1103.823,419.127,402.981,-179.583,18.970,152.034
C06842=1103.817,418.880,403.021,-179.585,18.962,152.032
C06843=1103.812,418.633,403.060,-179.587,18.954,152.031
C06844=1103.806,418.386,403.100,-179.589,18.946,152.029
C06845=1103.801,418.140,403.140,-179.591,18.938,152.028
C06846=1103.795,417.893,403.180,-179.594,18.930,152.026
C06847=1103.788,417.646,403.219,-179.596,18.922,152.024
C06848=1103.783,417.399,403.258,-179.598,18.914,152.023
C06849=1103.778,417.152,403.298,-179.599,18.907,152.021
C06850=1103.772,416.906,403.338,-179.601,18.899,152.020
C06851=1103.766,416.659,403.377,-179.603,18.891,152.018
C06852=1103.760,416.412,403.416,-179.605,18.884,152.017
C06853=1103.754,416.165,403.456,-179.608,18.876,152.015
C06854=1103.748,415.918,403.495,-179.610,18.868,152.014
C06855=1103.743,415.672,403.534,-179.611,18.861,152.012
C06856=1103.736,415.425,403.575,-179.614,18.854,152.011
C06857=1103.731,415.179,403.614,-179.616,18.846,152.009
C06858=1103.725,414.931,403.654,-179.618,18.838,152.008
C06859=1103.719,414.684,403.693,-179.620,18.831,152.006
C06860=1103.714,414.438,403.732,-179.622,18.824,152.005
C06861=1103.708,414.191,403.772,-179.624,18.816,152.003
C06862=1103.702,413.944,403.811,-179.626,18.809,152.002
C06863=1103.696,413.697,403.850,-179.629,18.801,152.000
C06864=1103.691,413.451,403.889,-179.630,18.795,151.999
C06865=1103.685,413.204,403.929,-179.632,18.787,151.997
C06866=1103.680,412.956,403.967,-179.635,18.780,151.996
C06867=1103.674,412.709,404.006,-179.636,18.773,151.994
C06868=1103.668,412.463,404.045,-179.639,18.765,151.993
C06869=1103.662,412.216,404.085,-179.641,18.758,151.992
C06870=1103.656,411.970,404.123,-179.643,18.751,151.990
C06871=1103.650,411.723,404.163,-179.645,18.744,151.989
C06872=1103.645,411.475,404.201,-179.647,18.736,151.987
C06873=1103.639,411.262,404.235,-179.650,18.730,151.986
C06874=1103.634,411.048,404.269,-179.651,18.724,151.985
C06875=1103.630,410.835,404.303,-179.653,18.718,151.984
C06876=1103.625,410.621,404.337,-179.654,18.712,151.983
C06877=1103.620,410.407,404.370,-179.656,18.706,151.981
C06878=1103.615,410.193,404.404,-179.658,18.700,151.980
C06879=1103.610,409.980,404.438,-179.660,18.694,151.979
C06880=1103.605,409.767,404.471,-179.662,18.687,151.978
C06881=1103.599,409.519,404.511,-179.664,18.681,151.977
C06882=1103.594,409.272,404.549,-179.666,18.674,151.975
C06883=1103.588,409.025,404.588,-179.669,18.666,151.974
C06884=1103.582,408.779,404.627,-179.671,18.660,151.973
C06885=1103.577,408.532,404.666,-179.673,18.653,151.971
C06886=1103.571,408.285,404.705,-179.675,18.646,151.970
C06887=1103.565,408.038,404.743,-179.678,18.639,151.969
C06888=1103.559,407.791,404.782,-179.679,18.633,151.967
C06889=1103.554,407.544,404.821,-179.682,18.626,151.966
C06890=1103.548,407.297,404.860,-179.684,18.619,151.965
C06891=1103.542,407.050,404.898,-179.686,18.612,151.964
C06892=1103.536,406.803,404.937,-179.688,18.606,151.962
C06893=1103.531,406.556,404.975,-179.691,18.599,151.961
C06894=1103.525,406.309,405.015,-179.692,18.592,151.960
C06895=1103.519,406.062,405.052,-179.695,18.586,151.959
C06896=1103.514,405.815,405.091,-179.697,18.579,151.957
C06897=1103.508,405.568,405.130,-179.700,18.572,151.956
C06898=1103.502,405.321,405.168,-179.702,18.566,151.955
C06899=1103.497,405.075,405.207,-179.704,18.559,151.954
C06900=1103.491,404.827,405.246,-179.706,18.553,151.953
C06901=1103.485,404.581,405.284,-179.709,18.546,151.951
C06902=1103.480,404.333,405.322,-179.711,18.540,151.950
C06903=1103.473,404.087,405.361,-179.713,18.534,151.949
C06904=1103.468,403.840,405.399,-179.716,18.527,151.948
C06905=1103.462,403.593,405.437,-179.717,18.521,151.947
C06906=1103.456,403.345,405.476,-179.720,18.514,151.946
C06907=1103.450,403.099,405.514,-179.722,18.508,151.944
C06908=1103.445,402.852,405.552,-179.724,18.502,151.943
C06909=1103.440,402.605,405.591,-179.727,18.495,151.942
C06910=1103.433,402.357,405.629,-179.729,18.489,151.941
C06911=1103.428,402.110,405.667,-179.732,18.483,151.940
C06912=1103.422,401.864,405.705,-179.734,18.477,151.939
C06913=1103.417,401.617,405.744,-179.736,18.471,151.938
C06914=1103.410,401.370,405.782,-179.739,18.464,151.936
C06915=1103.404,401.123,405.820,-179.741,18.458,151.935
C06916=1103.399,400.876,405.858,-179.743,18.452,151.934
C06917=1103.393,400.629,405.896,-179.746,18.446,151.933
C06918=1103.388,400.382,405.934,-179.748,18.439,151.932
C06919=1103.381,400.135,405.972,-179.750,18.434,151.931
C06920=1103.376,399.888,406.011,-179.752,18.428,151.930
C06921=1103.370,399.641,406.049,-179.755,18.421,151.929
C06922=1103.364,399.394,406.086,-179.757,18.415,151.928
C06923=1103.359,399.147,406.125,-179.759,18.409,151.927
C06924=1103.353,398.900,406.163,-179.762,18.404,151.926
C06925=1103.347,398.653,406.201,-179.764,18.397,151.925
C06926=1103.342,398.405,406.238,-179.767,18.392,151.924
C06927=1103.336,398.158,406.276,-179.769,18.386,151.923
C06928=1103.330,397.912,406.314,-179.771,18.380,151.922
C06929=1103.326,397.698,406.347,-179.773,18.375,151.921
C06930=1103.320,397.484,406.380,-179.775,18.370,151.920
C06931=1103.315,397.270,406.413,-179.777,18.364,151.919
C06932=1103.310,397.057,406.446,-179.780,18.359,151.918
C06933=1103.306,396.842,406.478,-179.782,18.354,151.917
C06934=1103.300,396.629,406.510,-179.784,18.349,151.916
C06935=1103.295,396.416,406.543,-179.786,18.344,151.916
C06936=1103.291,396.202,406.576,-179.788,18.339,151.915
C06937=1103.285,395.954,406.613,-179.791,18.333,151.914
C06938=1103.279,395.708,406.651,-179.793,18.328,151.913
C06939=1103.273,395.461,406.689,-179.795,18.322,151.912
C06940=1103.267,395.214,406.727,-179.797,18.317,151.911
C06941=1103.263,394.966,406.764,-179.800,18.311,151.910
C06942=1103.257,394.720,406.802,-179.803,18.305,151.909
C06943=1103.251,394.473,406.840,-179.805,18.299,151.908
C06944=1103.245,394.225,406.877,-179.807,18.294,151.907
C06945=1103.239,393.978,406.915,-179.810,18.288,151.906
C06946=1103.233,393.731,406.952,-179.812,18.283,151.905
C06947=1103.227,393.484,406.990,-179.814,18.277,151.904
C06948=1103.221,393.237,407.028,-179.817,18.272,151.903
C06949=1103.216,392.990,407.065,-179.819,18.266,151.902
C06950=1103.211,392.743,407.103,-179.822,18.260,151.902
C06951=1103.205,392.496,407.140,-179.825,18.255,151.901
C06952=1103.199,392.249,407.178,-179.827,18.249,151.900
C06953=1103.193,392.001,407.215,-179.830,18.244,151.899
C06954=1103.188,391.755,407.252,-179.832,18.239,151.898
C06955=1103.181,391.508,407.289,-179.835,18.233,151.897
C06956=1103.176,391.260,407.326,-179.837,18.228,151.896
C06957=1103.170,391.014,407.364,-179.840,18.223,151.896
C06958=1103.164,390.766,407.401,-179.842,18.217,151.895
C06959=1103.158,390.519,407.439,-179.845,18.212,151.894
C06960=1103.153,390.272,407.476,-179.847,18.207,151.893
C06961=1103.147,390.025,407.513,-179.850,18.201,151.892
C06962=1103.141,389.778,407.550,-179.853,18.196,151.892
C06963=1103.135,389.531,407.587,-179.855,18.190,151.891
C06964=1103.129,389.285,407.624,-179.858,18.185,151.890
C06965=1103.124,389.038,407.661,-179.860,18.180,151.889
C06966=1103.118,388.790,407.698,-179.863,18.175,151.888
C06967=1103.113,388.543,407.735,-179.865,18.170,151.887
C06968=1103.107,388.296,407.773,-179.868,18.165,151.887
C06969=1103.101,388.049,407.810,-179.871,18.159,151.886
C06970=1103.095,387.802,407.847,-179.873,18.154,151.885
C06971=1103.089,387.554,407.884,-179.876,18.149,151.884
C06972=1103.083,387.308,407.921,-179.878,18.144,151.883
C06973=1103.078,387.061,407.958,-179.881,18.139,151.883
C06974=1103.073,386.813,407.995,-179.883,18.134,151.882
C06975=1103.066,386.566,408.032,-179.886,18.128,151.881
C06976=1103.061,386.319,408.069,-179.889,18.123,151.880
C06977=1103.055,386.072,408.106,-179.891,18.118,151.880
C06978=1103.050,385.824,408.143,-179.894,18.114,151.879
C06979=1103.044,385.578,408.179,-179.897,18.108,151.878
C06980=1103.038,385.331,408.216,-179.899,18.103,151.877
C06981=1103.033,385.083,408.253,-179.902,18.098,151.877
C06982=1103.027,384.836,408.290,-179.904,18.093,151.876
C06983=1103.021,384.589,408.326,-179.907,18.088,151.875
C06984=1103.016,384.342,408.363,-179.910,18.083,151.875
C06985=1103.006,383.927,408.425,-179.914,18.075,151.873
C06986=1102.997,383.512,408.487,-179.918,18.067,151.872
C06987=1102.987,383.096,408.549,-179.923,18.058,151.871
C06988=1102.977,382.682,408.611,-179.928,18.050,151.870
C06989=1102.972,382.434,408.647,-179.930,18.045,151.869
C06990=1102.966,382.187,408.683,-179.933,18.041,151.868
C06991=1102.960,381.940,408.720,-179.936,18.036,151.868
C06992=1102.954,381.693,408.756,-179.938,18.031,151.867
C06993=1102.948,381.445,408.793,-179.941,18.027,151.866
C06994=1102.943,381.199,408.830,-179.943,18.022,151.866
C06995=1102.937,380.951,408.866,-179.946,18.017,151.865
C06996=1102.931,380.704,408.902,-179.949,18.013,151.865
C06997=1102.925,380.457,408.939,-179.952,18.007,151.864
C06998=1102.920,380.210,408.975,-179.955,18.003,151.863
C06999=1102.914,379.962,409.012,-179.957,17.998,151.863
C07000=1102.908,379.715,409.048,-179.960,17.993,151.862
C07001=1102.902,379.468,409.085,-179.962,17.989,151.861
C07002=1102.897,379.221,409.121,-179.965,17.985,151.861
C07003=1102.891,378.974,409.157,-179.968,17.980,151.860
C07004=1102.885,378.726,409.194,-179.971,17.975,151.860
C07005=1102.880,378.480,409.229,-179.974,17.970,151.859
C07006=1102.874,378.232,409.267,-179.977,17.966,151.858
C07007=1102.868,377.984,409.302,-179.979,17.962,151.858
C07008=1102.863,377.738,409.339,-179.981,17.957,151.857
C07009=1102.857,377.490,409.375,-179.985,17.953,151.857
C07010=1102.851,377.243,409.411,-179.987,17.948,151.856
C07011=1102.846,376.996,409.447,-179.990,17.943,151.856
C07012=1102.840,376.749,409.483,-179.993,17.938,151.855
C07013=1102.834,376.501,409.519,-179.995,17.934,151.854
C07014=1102.829,376.254,409.556,-179.998,17.930,151.854
C07015=1102.823,376.007,409.592,179.999,17.925,151.853
C07016=1102.818,375.760,409.628,179.996,17.921,151.853
C07017=1102.812,375.512,409.664,179.993,17.916,151.852
C07018=1102.806,375.265,409.700,179.991,17.912,151.852
C07019=1102.801,375.018,409.736,179.988,17.907,151.851
C07020=1102.795,374.770,409.772,179.985,17.903,151.851
C07021=1102.789,374.523,409.808,179.982,17.898,151.850
C07022=1102.783,374.276,409.845,179.980,17.895,151.849
C07023=1102.777,374.028,409.880,179.977,17.890,151.849
C07024=1102.772,373.781,409.916,179.974,17.886,151.848
C07025=1102.766,373.534,409.952,179.971,17.881,151.848
C07026=1102.760,373.287,409.988,179.969,17.877,151.847
C07027=1102.754,373.040,410.023,179.965,17.873,151.847
C07028=1102.748,372.792,410.059,179.962,17.869,151.846
C07029=1102.743,372.545,410.096,179.959,17.864,151.846
C07030=1102.737,372.298,410.131,179.957,17.861,151.845
C07031=1102.731,372.050,410.167,179.954,17.856,151.845
C07032=1102.726,371.803,410.202,179.951,17.852,151.844
C07033=1102.720,371.555,410.238,179.949,17.848,151.844
C07034=1102.714,371.308,410.274,179.946,17.844,151.844
C07035=1102.708,371.061,410.310,179.942,17.839,151.843
C07036=1102.702,370.814,410.345,179.939,17.835,151.843
C07037=1102.694,370.425,410.402,179.935,17.829,151.842
C07038=1102.685,370.037,410.457,179.931,17.822,151.841
C07039=1102.676,369.649,410.513,179.926,17.816,151.840
C07040=1102.667,369.261,410.569,179.922,17.809,151.840
C07041=1102.662,369.013,410.605,179.919,17.805,151.839
C07042=1102.656,368.766,410.640,179.916,17.801,151.839
C07043=1102.650,368.518,410.676,179.913,17.797,151.838
C07044=1102.645,368.271,410.711,179.910,17.793,151.838
C07045=1102.639,368.024,410.747,179.907,17.789,151.838
C07046=1102.633,367.777,410.783,179.904,17.785,151.837
C07047=1102.627,367.529,410.818,179.901,17.781,151.837
C07048=1102.622,367.282,410.854,179.899,17.777,151.836
C07049=1102.616,367.034,410.889,179.896,17.773,151.836
C07050=1102.611,366.787,410.924,179.892,17.769,151.835
C07051=1102.605,366.540,410.959,179.890,17.765,151.835
C07052=1102.599,366.292,410.995,179.887,17.761,151.835
C07053=1102.594,366.045,411.031,179.884,17.757,151.834
C07054=1102.588,365.797,411.066,179.881,17.753,151.834
C07055=1102.582,365.550,411.100,179.878,17.749,151.834
C07056=1102.576,365.302,411.136,179.876,17.746,151.833
C07057=1102.570,365.055,411.171,179.872,17.742,151.833
C07058=1102.565,364.807,411.206,179.869,17.737,151.832
C07059=1102.559,364.560,411.242,179.867,17.734,151.832
C07060=1102.554,364.313,411.277,179.863,17.730,151.832
C07061=1102.547,364.065,411.312,179.861,17.726,151.831
C07062=1102.542,363.818,411.347,179.858,17.722,151.831
C07063=1102.536,363.571,411.383,179.854,17.718,151.831
C07064=1102.531,363.323,411.417,179.852,17.715,151.830
C07065=1102.525,363.075,411.453,179.848,17.711,151.830
C07066=1102.519,362.828,411.487,179.846,17.707,151.829
C07067=1102.513,362.581,411.522,179.843,17.703,151.829
C07068=1102.507,362.333,411.558,179.840,17.700,151.829
C07069=1102.502,362.086,411.593,179.837,17.696,151.829
C07070=1102.496,361.839,411.628,179.833,17.692,151.828
C07071=1102.490,361.591,411.663,179.831,17.688,151.828
C07072=1102.485,361.344,411.698,179.828,17.685,151.828
C07073=1102.478,361.096,411.732,179.825,17.681,151.827
C07074=1102.473,360.849,411.768,179.822,17.677,151.827
C07075=1102.468,360.601,411.802,179.819,17.674,151.827
C07076=1102.462,360.353,411.837,179.816,17.670,151.826
C07077=1102.456,360.106,411.872,179.813,17.667,151.826
C07078=1102.451,359.859,411.907,179.810,17.663,151.826
C07079=1102.444,359.611,411.942,179.807,17.660,151.825
C07080=1102.439,359.364,411.977,179.804,17.656,151.825
C07081=1102.434,359.116,412.011,179.801,17.652,151.825
C07082=1102.427,358.869,412.046,179.798,17.649,151.825
C07083=1102.422,358.621,412.081,179.795,17.645,151.824
C07084=1102.416,358.374,412.115,179.792,17.641,151.824
C07085=1102.410,358.126,412.151,179.789,17.637,151.824
C07086=1102.405,357.879,412.185,179.786,17.634,151.824
C07087=1102.399,357.631,412.220,179.782,17.631,151.823
C07088=1102.394,357.384,412.254,179.780,17.627,151.823
C07089=1102.384,357.010,412.307,179.775,17.622,151.822
C07090=1102.376,356.637,412.359,179.770,17.617,151.822
C07091=1102.367,356.263,412.411,179.766,17.612,151.822
C07092=1102.359,355.890,412.463,179.761,17.606,151.821
C07093=1102.353,355.643,412.497,179.758,17.603,151.821
C07094=1102.348,355.395,412.532,179.756,17.599,151.821
C07095=1102.342,355.148,412.566,179.752,17.596,151.821
C07096=1102.336,354.900,412.601,179.749,17.592,151.820
C07097=1102.330,354.653,412.636,179.747,17.589,151.820
C07098=1102.325,354.405,412.670,179.743,17.586,151.820
C07099=1102.319,354.158,412.704,179.740,17.582,151.820
C07100=1102.314,353.910,412.739,179.737,17.579,151.820
C07101=1102.307,353.662,412.773,179.734,17.575,151.819
C07102=1102.302,353.415,412.808,179.731,17.572,151.819
C07103=1102.296,353.168,412.842,179.728,17.569,151.819
C07104=1102.291,352.920,412.876,179.724,17.565,151.819
C07105=1102.285,352.672,412.911,179.722,17.562,151.819
C07106=1102.279,352.424,412.945,179.719,17.559,151.818
C07107=1102.273,352.177,412.979,179.715,17.555,151.818
C07108=1102.268,351.929,413.013,179.713,17.552,151.818
C07109=1102.262,351.682,413.047,179.709,17.549,151.818
C07110=1102.256,351.434,413.082,179.706,17.546,151.818
C07111=1102.250,351.187,413.116,179.703,17.542,151.817
C07112=1102.245,350.939,413.150,179.700,17.539,151.817
C07113=1102.239,350.692,413.185,179.697,17.536,151.817
C07114=1102.234,350.444,413.218,179.694,17.533,151.817
C07115=1102.228,350.196,413.253,179.691,17.530,151.817
C07116=1102.223,349.949,413.287,179.687,17.526,151.816
C07117=1102.216,349.701,413.321,179.684,17.523,151.816
C07118=1102.211,349.453,413.354,179.682,17.520,151.816
C07119=1102.205,349.205,413.389,179.678,17.516,151.816
C07120=1102.200,348.958,413.423,179.675,17.513,151.816
C07121=1102.194,348.710,413.456,179.672,17.511,151.816
C07122=1102.188,348.463,413.490,179.669,17.507,151.816
C07123=1102.182,348.216,413.524,179.666,17.504,151.815
C07124=1102.178,347.968,413.558,179.662,17.500,151.815
C07125=1102.171,347.720,413.593,179.660,17.497,151.815
C07126=1102.165,347.472,413.627,179.657,17.494,151.815
C07127=1102.160,347.224,413.660,179.653,17.491,151.815
C07128=1102.154,346.977,413.694,179.650,17.488,151.815
C07129=1102.148,346.729,413.728,179.647,17.485,151.814
C07130=1102.142,346.482,413.762,179.644,17.482,151.814
C07131=1102.137,346.234,413.796,179.641,17.479,151.814
C07132=1102.132,345.986,413.830,179.638,17.476,151.814
C07133=1102.126,345.739,413.864,179.634,17.473,151.814
C07134=1102.120,345.491,413.897,179.631,17.470,151.814
C07135=1102.114,345.244,413.931,179.628,17.467,151.814
C07136=1102.109,344.996,413.964,179.625,17.463,151.814
C07137=1102.103,344.748,413.998,179.622,17.461,151.814
C07138=1102.097,344.501,414.032,179.619,17.458,151.814
C07139=1102.092,344.253,414.065,179.615,17.455,151.813
C07140=1102.086,344.006,414.099,179.612,17.452,151.813
C07141=1102.077,343.634,414.150,179.608,17.448,151.813
C07142=1102.069,343.263,414.200,179.603,17.443,151.813
C07143=1102.060,342.892,414.250,179.598,17.439,151.813
C07144=1102.052,342.521,414.300,179.593,17.434,151.813
C07145=1102.046,342.273,414.334,179.590,17.431,151.813
C07146=1102.041,342.025,414.367,179.587,17.429,151.813
C07147=1102.035,341.778,414.401,179.583,17.425,151.813
C07148=1102.029,341.530,414.434,179.581,17.422,151.812
C07149=1102.024,341.282,414.468,179.577,17.420,151.812
C07150=1102.018,341.034,414.501,179.575,17.417,151.812
C07151=1102.012,340.786,414.534,179.571,17.414,151.812
C07152=1102.006,340.539,414.568,179.568,17.411,151.812
C07153=1102.000,340.292,414.601,179.565,17.408,151.812
C07154=1101.995,340.044,414.635,179.561,17.405,151.812
C07155=1101.989,339.796,414.668,179.558,17.402,151.812
C07156=1101.984,339.548,414.701,179.555,17.399,151.812
C07157=1101.978,339.300,414.735,179.552,17.397,151.812
C07158=1101.973,339.052,414.768,179.548,17.393,151.812
C07159=1101.966,338.805,414.801,179.545,17.391,151.812
C07160=1101.960,338.557,414.835,179.542,17.388,151.812
C07161=1101.955,338.309,414.868,179.539,17.386,151.812
C07162=1101.950,338.062,414.901,179.536,17.383,151.812
C07163=1101.944,337.814,414.934,179.532,17.380,151.812
C07164=1101.938,337.566,414.967,179.529,17.377,151.812
C07165=1101.932,337.319,415.000,179.526,17.375,151.812
C07166=1101.927,337.071,415.034,179.523,17.372,151.812
C07167=1101.921,336.823,415.067,179.519,17.369,151.812
C07168=1101.915,336.575,415.100,179.516,17.366,151.812
C07169=1101.910,336.327,415.133,179.513,17.364,151.812
C07170=1101.903,336.080,415.166,179.510,17.361,151.811
C07171=1101.898,335.831,415.199,179.507,17.358,151.812
C07172=1101.893,335.584,415.232,179.503,17.355,151.812
C07173=1101.887,335.336,415.264,179.500,17.353,151.812
C07174=1101.881,335.088,415.298,179.497,17.350,151.812
C07175=1101.876,334.841,415.331,179.494,17.347,151.811
C07176=1101.869,334.593,415.364,179.491,17.345,151.811
C07177=1101.864,334.345,415.397,179.487,17.342,151.811
C07178=1101.858,334.098,415.429,179.484,17.339,151.812
C07179=1101.853,333.850,415.462,179.481,17.337,151.812
C07180=1101.847,333.602,415.495,179.478,17.334,151.812
C07181=1101.841,333.354,415.528,179.475,17.332,151.812
C07182=1101.835,333.106,415.562,179.472,17.329,151.811
C07183=1101.830,332.859,415.593,179.468,17.326,151.811
C07184=1101.825,332.611,415.627,179.465,17.323,151.812
C07185=1101.819,332.363,415.660,179.462,17.321,151.812
C07186=1101.813,332.115,415.692,179.458,17.318,151.812
C07187=1101.807,331.867,415.725,179.455,17.316,151.812
C07188=1101.801,331.619,415.758,179.452,17.314,151.812
C07189=1101.796,331.372,415.790,179.448,17.311,151.812
C07190=1101.790,331.124,415.823,179.445,17.308,151.812
C07191=1101.784,330.876,415.856,179.442,17.306,151.812
C07192=1101.778,330.628,415.888,179.439,17.303,151.812
C07193=1101.770,330.251,415.938,179.434,17.300,151.812
C07194=1101.761,329.873,415.987,179.429,17.296,151.812
C07195=1101.752,329.496,416.037,179.423,17.292,151.812
C07196=1101.743,329.119,416.087,179.418,17.289,151.812
C07197=1101.737,328.872,416.119,179.415,17.286,151.812
C07198=1101.731,328.624,416.151,179.412,17.284,151.812
C07199=1101.726,328.375,416.184,179.409,17.281,151.812
C07200=1101.720,328.128,416.216,179.406,17.279,151.813
C07201=1101.714,327.880,416.248,179.403,17.277,151.813
C07202=1101.709,327.632,416.281,179.399,17.273,151.813
C07203=1101.703,327.384,416.313,179.395,17.271,151.813
C07204=1101.697,327.136,416.346,179.392,17.269,151.813
C07205=1101.692,326.889,416.378,179.389,17.266,151.813
C07206=1101.686,326.640,416.410,179.386,17.264,151.813
C07207=1101.680,326.393,416.443,179.382,17.262,151.813
C07208=1101.674,326.145,416.475,179.379,17.259,151.813
C07209=1101.669,325.897,416.507,179.376,17.257,151.813
C07210=1101.663,325.649,416.540,179.373,17.255,151.813
C07211=1101.657,325.402,416.572,179.370,17.252,151.813
C07212=1101.651,325.153,416.604,179.366,17.250,151.814
C07213=1101.645,324.906,416.637,179.363,17.248,151.814
C07214=1101.640,324.658,416.669,179.360,17.246,151.814
C07215=1101.634,324.410,416.701,179.356,17.243,151.814
C07216=1101.628,324.162,416.733,179.353,17.240,151.814
C07217=1101.623,323.915,416.765,179.349,17.238,151.814
C07218=1101.617,323.666,416.797,179.346,17.236,151.814
C07219=1101.612,323.419,416.830,179.343,17.234,151.814
C07220=1101.606,323.170,416.862,179.340,17.231,151.814
C07221=1101.600,322.922,416.894,179.336,17.229,151.814
C07222=1101.595,322.675,416.925,179.333,17.227,151.814
C07223=1101.588,322.427,416.958,179.330,17.224,151.815
C07224=1101.583,322.180,416.990,179.326,17.222,151.815
C07225=1101.578,321.931,417.022,179.323,17.220,151.815
C07226=1101.572,321.684,417.054,179.320,17.217,151.815
C07227=1101.566,321.435,417.086,179.317,17.215,151.815
C07228=1101.561,321.188,417.118,179.313,17.213,151.815
C07229=1101.555,320.940,417.150,179.310,17.211,151.815
C07230=1101.549,320.691,417.182,179.307,17.208,151.815
C07231=1101.544,320.444,417.213,179.303,17.206,151.816
C07232=1101.538,320.196,417.245,179.300,17.204,151.816
C07233=1101.532,319.948,417.277,179.297,17.202,151.816
C07234=1101.527,319.700,417.310,179.293,17.200,151.816
C07235=1101.522,319.452,417.341,179.290,17.197,151.816
C07236=1101.516,319.204,417.373,179.287,17.195,151.816
C07237=1101.510,318.956,417.405,179.284,17.193,151.816
C07238=1101.505,318.709,417.437,179.280,17.191,151.816
C07239=1101.499,318.461,417.469,179.277,17.189,151.817
C07240=1101.494,318.212,417.500,179.274,17.186,151.817
C07241=1101.488,317.964,417.532,179.270,17.184,151.817
C07242=1101.482,317.717,417.563,179.267,17.182,151.817
C07243=1101.477,317.469,417.595,179.264,17.179,151.817
C07244=1101.471,317.221,417.627,179.260,17.177,151.817
C07245=1101.462,316.836,417.676,179.256,17.174,151.817
C07246=1101.454,316.453,417.725,179.250,17.170,151.818
C07247=1101.445,316.068,417.774,179.245,17.167,151.818
C07248=1101.437,315.683,417.823,179.240,17.164,151.818
C07249=1101.432,315.436,417.855,179.236,17.162,151.818
C07250=1101.425,315.188,417.886,179.233,17.160,151.818
C07251=1101.420,314.940,417.917,179.230,17.157,151.819
C07252=1101.414,314.691,417.949,179.226,17.155,151.819
C07253=1101.408,314.444,417.981,179.223,17.153,151.819
C07254=1101.403,314.196,418.011,179.219,17.151,151.819
C07255=1101.397,313.948,418.043,179.216,17.149,151.819
C07256=1101.391,313.700,418.075,179.212,17.147,151.820
C07257=1101.385,313.452,418.106,179.209,17.145,151.820
C07258=1101.379,313.204,418.137,179.206,17.143,151.820
C07259=1101.373,312.956,418.169,179.203,17.142,151.820
